# B&R Automation Studio project ACOPOStrak (part 2)

### Config_1.assembly - 5PC900_TS17_00/mappMotion/TrakOval/Config_1.assembly
```
Element gAssembly_1 (Type=assembly)
  Tracks:
    TrackSeparation = 0.030
    Track[1]:
      Segments:
        SegmentRef[1] = ::Seg_A_1
        SegmentRef[2] = ::Seg_A_2
        SegmentRef[3] = ::Seg_A_3
        SegmentRef[4] = ::Seg_A_4
        SegmentRef[5] = ::Seg_A_5
        SegmentRef[6] = ::Seg_A_6
        SegmentRef[7] = ::Seg_A_7
        SegmentRef[8] = ::Seg_A_8
        SegmentRef[9] = ::Seg_A_9
        SegmentRef[10] = ::Seg_A_10
        SegmentRef[11] = ::Seg_A_11
        SegmentRef[12] = ::Seg_A_12
        SegmentRef[13] = ::Seg_A_13
      Position = Absolute
        SegmentRef = ::Seg_A_1
        SegmentCountDirection = RightToLeft
        Translation:
          X = 0.0
          Y = 0.0
          Z = 0.0
        Orientation:
          Angle1 = 0.0
          Angle2 = 0.0
          Angle3 = 180
    Track[2]:
      Segments:
        SegmentRef[1] = ::Seg_A_14
        SegmentRef[2] = ::Seg_A_15
        SegmentRef[3] = ::Seg_A_16
        SegmentRef[4] = ::Seg_A_17
        SegmentRef[5] = ::Seg_A_18
        SegmentRef[6] = ::Seg_A_19
        SegmentRef[7] = ::Seg_A_20
        SegmentRef[8] = ::Seg_A_21
        SegmentRef[9] = ::Seg_A_22
        SegmentRef[10] = ::Seg_A_23
        SegmentRef[11] = ::Seg_A_24
        SegmentRef[12] = ::Seg_A_25
        SegmentRef[13] = ::Seg_A_26
      Position = Absolute
        SegmentRef = ::Seg_A_14
        SegmentCountDirection = RightToLeft
        Translation:
          X = 0.0
          Y = 0.0
          Z = 0.0
        Orientation:
          Angle1 = 0.0
          Angle2 = 0.0
          Angle3 = 0.0
    Track[3]:
      Segments:
        SegmentRef[1] = ::Seg_B_1
        SegmentRef[2] = :Seg_B_2
      Position = Absolute
        SegmentRef = :Seg_B_1
        SegmentCountDirection = RightToLeft
        Translation:
          X = 0.0
          Y = 0.0
          Z = 0.0
        Orientation:
          Angle1 = 0.0
          Angle2 = 0.0
          Angle3 = 0.0
    Track[4]:
      Segments:
        SegmentRef[1] = :Seg_B_3
        SegmentRef[2] = :Seg_B_4
        SegmentRef[3] = :Seg_B_5
      Position = Absolute
        SegmentRef = :Seg_B_3
        SegmentCountDirection = RightToLeft
        Translation:
          X = 0.0
          Y = 0.0
          Z = 0.0
        Orientation:
          Angle1 = 0.0
          Angle2 = 0.0
          Angle3 = 0.0
    Track[5]:
      Segments:
        SegmentRef[1] = :Seg_B_6
        SegmentRef[2] = :Seg_B_7
      Position = Absolute
        SegmentRef = :Seg_B_6
        SegmentCountDirection = RightToLeft
        Translation:
          X = 0.0
          Y = 0.0
          Z = 0.0
        Orientation:
          Angle1 = 0.0
          Angle2 = 0.0
          Angle3 = 0.0
  CommonSegmentSettings:
    SegmentSimulationOnPLC = Off
    StopReaction = InductionHalt
    SpeedFilter = NotUsed
    ControllerParameters:
      DefaultParameter:
        Controller:
          Position:
            ProportionalGain = 200
          Speed:
            ProportionalGain = 80
            IntegrationTime = 0.0
          FeedForward:
            TotalMass = 1
            ForcePositive = 0.0
            ForceNegative = 0.0
            SpeedForceFactor = 0.0
            ForceLoad = 0.0
        MovementErrorLimits:
          PositionError = 0.001
          VelocityError = 0.05
      AdditionalParameterSets = NotUsed
  Shuttles:
    MaxShuttleCount = 25
    ShuttleStereotypes:
      ShuttleStRef[1] = ShuttleStereotype_1
    MagnetPlateConfigurations:
      ShuttleType[1] = 8F1SA.100.xxxxxx-x
    CollisionAvoidance:
      Strategy = Constant
      MaximumModelDimensions:
        Length:
          ExtentToFront = 0.025
          ExtentToBack = 0.025
        Width:
          Width = 0.040
  Visualization:
    MonitoringPv = gShuttleMon
    ProcessingTaskClass = 1
```

### Config_2.shuttlestereotype - 5PC900_TS17_00/mappMotion/TrakOval/Config_2.shuttlestereotype
```
Element ShuttleStereotype_1 (Type=shuttlestereotype)
  MeasurementUnit = 5067858
  MeasurementResolution = 0.00001
  MovementLimits = Internal
    VelocityIsReadOnly = 0
    Velocity:
      Velocity = 4
    AccelerationIsReadOnly = 0
    Acceleration:
      Acceleration = 40
    DecelerationIsReadOnly = 0
    Deceleration:
      Deceleration = 40
  JerkFilter = NotUsed
  UserData:
    Size = 12
```

### Config_3.sector - 5PC900_TS17_00/mappMotion/TrakOval/Config_3.sector
```
Element SectorTrackA (Type=sector)
  Type = Composed
    StartSegment:
      SegmentRef = ::Seg_A_1
    IntermediateSegments:
      SegmentRef[1] = ::Seg_A_2
      SegmentRef[2] = ::Seg_A_3
      SegmentRef[3] = ::Seg_A_4
      SegmentRef[4] = ::Seg_A_5
      SegmentRef[5] = ::Seg_A_6
      SegmentRef[6] = ::Seg_A_7
      SegmentRef[7] = ::Seg_A_8
      SegmentRef[8] = ::Seg_A_9
      SegmentRef[9] = ::Seg_A_10
      SegmentRef[10] = ::Seg_A_11
      SegmentRef[11] = ::Seg_A_12
      SegmentRef[12] = ::Seg_A_13
      SegmentRef[13] = ::Seg_A_14
      SegmentRef[14] = ::Seg_A_15
      SegmentRef[15] = ::Seg_A_16
      SegmentRef[16] = ::Seg_A_17
      SegmentRef[17] = ::Seg_A_18
      SegmentRef[18] = ::Seg_A_19
      SegmentRef[19] = ::Seg_A_20
      SegmentRef[20] = ::Seg_A_21
      SegmentRef[21] = ::Seg_A_22
      SegmentRef[22] = ::Seg_A_23
      SegmentRef[23] = ::Seg_A_24
      SegmentRef[24] = ::Seg_A_25
    EndSegment:
      SegmentRef = ::Seg_A_26
      PositionRelativeTo = FromEnd
Element SectorPouring_1 (Type=sector)
  Type = Subsector
    SectorRef = SectorTrackA
    Start:
      Position = 0.33
    Length = 0.1
    Direction = Positive
```

### Config_5.assembly - 5PC900_TS17_00/mappMotion/TrakOval/Config_5.assembly
```
Element gAssembly_1 (Type=assembly)
  Tracks:
    TrackSeparation = 0.030
    Track[1]:
      Segments:
        SegmentRef[1] = ::Seg_A_1
        SegmentRef[2] = ::Seg_A_2
        SegmentRef[3] = ::Seg_A_3
        SegmentRef[4] = ::Seg_A_4
        SegmentRef[5] = ::Seg_A_5
        SegmentRef[6] = ::Seg_A_6
        SegmentRef[7] = ::Seg_A_7
        SegmentRef[8] = ::Seg_A_8
        SegmentRef[9] = ::Seg_A_9
        SegmentRef[10] = ::Seg_A_10
        SegmentRef[11] = ::Seg_A_11
        SegmentRef[12] = ::Seg_A_12
        SegmentRef[13] = ::Seg_A_13
        SegmentRef[14] = ::Seg_A_14
        SegmentRef[15] = ::Seg_A_15
        SegmentRef[16] = ::Seg_A_16
        SegmentRef[17] = ::Seg_A_17
        SegmentRef[18] = ::Seg_A_18
        SegmentRef[19] = ::Seg_A_19
        SegmentRef[20] = ::Seg_A_20
        SegmentRef[21] = ::Seg_A_21
        SegmentRef[22] = ::Seg_A_22
        SegmentRef[23] = ::Seg_A_23
        SegmentRef[24] = ::Seg_A_24
        SegmentRef[25] = ::Seg_A_25
        SegmentRef[26] = ::Seg_A_26
      Position = Absolute
        SegmentRef = ::Seg_A_1
        SegmentCountDirection = RightToLeft
        Translation:
          X = 0.0
          Y = 0.0
          Z = 0.0
        Orientation:
          Angle1 = 0.0
          Angle2 = 0.0
          Angle3 = 180
    Track[2]:
      Segments:
        SegmentRef[1] = ::Seg_B_3
        SegmentRef[2] = ::Seg_B_2
        SegmentRef[3] = ::Seg_B_1
      Position = RelativeToOne
        TrackSegmentPosition:
          SegmentRef = ::Seg_B_1
          Position = 0
          PositionRelativeTo = FromEnd
        Base:
          SegmentRef = ::Seg_A_1
          Position = 0.1
    Track[3]:
      Segments:
        SegmentRef[1] = ::Seg_B_4
        SegmentRef[2] = ::Seg_B_5
        SegmentRef[3] = ::Seg_B_6
        SegmentRef[4] = ::Seg_B_7
        SegmentRef[5] = ::Seg_B_8
      Position = RelativeToOne
        TrackSegmentPosition:
          SegmentRef = ::Seg_B_4
        Base:
          SegmentRef = ::Seg_B_3
          Position = 0.33
    Track[4]:
      Segments:
        SegmentRef[1] = ::Seg_B_11
        SegmentRef[2] = ::Seg_B_10
        SegmentRef[3] = ::Seg_B_9
      Position = RelativeToTwo
        AlignmentToFirst:
          SegmentRefNewFirst = ::Seg_B_11
          SegmentRefBaseFirst = ::Seg_A_7
        AlignmentToSecond:
          SegmentRefNewSecond = ::Seg_B_9
          SegmentRefBaseSecond = ::Seg_B_8
  CommonSegmentSettings:
    SegmentSimulationOnPLC = Off
    StopReaction = InductionHalt
    SpeedFilter = NotUsed
    ControllerParameters:
      DefaultParameter:
        Controller:
          Position:
            ProportionalGain = 200
          Speed:
            ProportionalGain = 80
            IntegrationTime = 0.0
          FeedForward:
            TotalMass = 1
            ForcePositive = 0.0
            ForceNegative = 0.0
            SpeedForceFactor = 0.0
            ForceLoad = 0.0
        MovementErrorLimits:
          PositionError = 0.001
          VelocityError = 0.05
      AdditionalParameterSets = NotUsed
  Shuttles:
    MaxShuttleCount = 25
    ShuttleStereotypes:
      ShuttleStRef[1] = ShuttleStereotype_1
    MagnetPlateConfigurations:
      ShuttleType[1] = 8F1SA.100.xxxxxx-x
    CollisionAvoidance:
      Strategy = Constant
      MaximumModelDimensions:
        Length:
          ExtentToFront = 0.025
          ExtentToBack = 0.025
        Width:
          Width = 0.040
  Visualization:
    MonitoringPv = gShuttleMon
    ProcessingTaskClass = 1
```

### Config_7.sector - 5PC900_TS17_00/mappMotion/TrakOval/Config_7.sector
```
Element SectorTrackA (Type=sector)
  Type = Composed
    StartSegment:
      SegmentRef = ::Seg_A_1
    IntermediateSegments:
      SegmentRef[1] = ::Seg_A_2
      SegmentRef[2] = ::Seg_A_3
      SegmentRef[3] = ::Seg_A_4
      SegmentRef[4] = ::Seg_A_5
      SegmentRef[5] = ::Seg_A_6
      SegmentRef[6] = ::Seg_A_7
      SegmentRef[7] = ::Seg_A_8
      SegmentRef[8] = ::Seg_A_9
      SegmentRef[9] = ::Seg_A_10
      SegmentRef[10] = ::Seg_A_11
      SegmentRef[11] = ::Seg_A_12
      SegmentRef[12] = ::Seg_A_13
      SegmentRef[13] = ::Seg_A_14
      SegmentRef[14] = ::Seg_A_15
      SegmentRef[15] = ::Seg_A_16
      SegmentRef[16] = ::Seg_A_17
      SegmentRef[17] = ::Seg_A_18
      SegmentRef[18] = ::Seg_A_19
      SegmentRef[19] = ::Seg_A_20
      SegmentRef[20] = ::Seg_A_21
      SegmentRef[21] = ::Seg_A_22
      SegmentRef[22] = ::Seg_A_23
      SegmentRef[23] = ::Seg_A_24
      SegmentRef[24] = ::Seg_A_25
    EndSegment:
      SegmentRef = ::Seg_A_26
      PositionRelativeTo = FromEnd
```

### Alarm.mpalarmxcore - 5PC900_TS17_00/mappServices/Alarm.mpalarmxcore
```
Element gAlarmXCore (Type=mpalarmxcore)
  mapp.AlarmX.Core.Configuration:
    [0]:
      Name = InterruptAlarm
      Message = Procces was interrupted
    [1]:
      Name = SectorTopAlarm
      Message = Top Pouring Sector inefficient
      Code = 1
      Behavior = DiscreteValueMonitoring
        Monitoring:
          MonitoredPV = ::TrakMoveme:VisPouring_Top_Broken
          TriggerValues:
            [0] = FALSE
    [2]:
      Name = SectorDownAlarm
      Message = Down Pouring Sector inefficient
      Code = 2
      Behavior = DiscreteValueMonitoring
        Monitoring:
          MonitoredPV = ::TrakMoveme:VisPouring_Down_Broken
          TriggerValues:
            [0] = FALSE
    [3]:
      Name = SuddenlyStopAlarm
      Message = Procces was suddenly stopped
    [4]:
      Name = SectorCappingAlarm
      Message = Capping Sector inefficient
      Code = 3
      Behavior = DiscreteValueMonitoring
        Monitoring:
          MonitoredPV = ::TrakMoveme:VisCapping_Broken
          TriggerValues:
            [0] = FALSE
    [5]:
      Name = SectorInputAlarm
      Message = Input Sector inefficient
      Code = 4
      Behavior = DiscreteValueMonitoring
        Monitoring:
          MonitoredPV = ::gVisInput_Broken
          TriggerValues:
            [0] = FALSE
    [6]:
      Name = SectorIOutputAlarm
      Message = Output Sector inefficient
      Code = 5
      Behavior = DiscreteValueMonitoring
        Monitoring:
          MonitoredPV = ::gVisOutput_Broken
          TriggerValues:
            [0] = FALSE
    [7]:
      Name = ManualWorkAlarm
      Message = Trak is in manual work
      Code = 6
      Severity = 10
      Behavior = DiscreteValueMonitoring
        Monitoring:
          MonitoredPV = ::TrakMoveme:VisManual
          TriggerValues:
            [0] = TRUE
    [8]:
      Name = HighAccelerationAlarm
      Message = High acceleration has been set
      Code = 7
      Severity = 10
      Behavior = LevelMonitoring
        Monitoring:
          MonitoredPV = ::TrakMoveme:VisAcceleration
          HighLimitEnable = Static
            Limit = 37
            LimitText = High acceleration has been set
    [9]:
      Name = HighDecelerationAlarm
      Message = High deceleration has been set
      Code = 9
      Severity = 10
      Behavior = LevelMonitoring
        Monitoring:
          MonitoredPV = ::TrakMoveme:VisDeceleration
          HighLimitEnable = Static
            Limit = 37
            LimitText = High deceleration has been set
    [10]:
      Name = HighVelocityAlarm
      Message = High velocity has been set
      Code = 10
      Severity = 10
      Behavior = LevelMonitoring
        Monitoring:
          MonitoredPV = ::TrakMoveme:VisVelocity
          HighLimitEnable = Static
            Limit = 3.5
            LimitText = High velocity has been set
```

## Logical view

Binary libraries used (declarations not repeated): operator, runtime, astime, AsIecCon, CoTrace, AsZip, FileIO, McBase, McAxis, McAcpTrak 5.10.1, AsBrStr, MpRobotics 5.10.1, MpBase, McAxGroup, McPathGen, McProgInt, McAcpAx, MpRecipe 5.10.1, standard, sys_lib, MpAlarmX, MpFile 5.10.1, MpServer

### Global.typ - Global data types
```iecst
(*shuttle-UserData structure*)

TYPE
	ShuttleUserData_typ : 	STRUCT
		Color : ShuttleColor_enum; (*example: product colour*)
		Weight : REAL; (*example: product weight*)
		Partnumber : UDINT; (*example: product part number*)
	END_STRUCT;
	ShuttleColor_enum :
		(
		ORANGE,
		GREEN,
		RED,
		BLUE,
		WHITE
		);
END_TYPE

(*Assembly Interface Type*)

TYPE
	TrakAsmCommand_type : 	STRUCT
		Power : BOOL;
		ShuttleStart : BOOL;
		ShuttleStop : BOOL;
	END_STRUCT;
	TrakAsmParameter_type : 	STRUCT
		Velocity : REAL;
		Acceleration : REAL;
		Deceleration : REAL;
	END_STRUCT;
	TrakAsmStatus_type : 	STRUCT
		Disabled : BOOL;
		Ready : BOOL;
		Homing : BOOL;
		Stopping : BOOL;
		ErrorStop : BOOL;
	END_STRUCT;
	TrakAsm_type : 	STRUCT
		Command : TrakAsmCommand_type;
		Parameter : TrakAsmParameter_type;
		Status : TrakAsmStatus_type;
	END_STRUCT;
	Order_type : 	STRUCT
		numberOfPackages : USINT := 5;
		bottlesPerPackage : USINT := 5;
		bottleSize : BottleSize_enum := BOTTLE_SIZE_LARGE;
		drinkColor : DrinkColor_enum := DRINK_COLOR_RED;
	END_STRUCT;
	DrinkColor_enum :
		(
		DRINK_COLOR_RED,
		DRINK_COLOR_GREEN,
		DRINK_COLOR_BLUE
		);
	BottleSize_enum :
		(
		BOTTLE_SIZE_LARGE,
		BOTTLE_SIZE_SMALL
		);
END_TYPE
```

### Global.var - Global variables
```iecst
VAR
	VisManual : BOOL;
	gbottlesDone : BOOL;
	gPartyOn : BOOL;
	gVisTurn_Broken : BOOL;
	ShuttleNumber : USINT;
END_VAR
(*Assembly interface*)
VAR
	gBottleInPlace_Turn : BOOL;
	gShuttleInPlace_Turn : BOOL;
	gTrakAsm : TrakAsm_type;
END_VAR
(*shuttle-UserData structure*)
VAR
	gShuttleUserData : ShuttleUserData_typ;
END_VAR
(*shuttle monitor structure for Vis*)
VAR
	gShuttleMon : McAcpTrakAssemblyMonData;
END_VAR
(*Bottle input and output*)
VAR
	gBottleInPlace_Input : BOOL := FALSE;
	gBottleInPlace_Output : BOOL := FALSE;
	gShuttleInPlace_Output : BOOL := FALSE;
	gShuttleInPlace_Input : BOOL := FALSE;
END_VAR
(*Trak Variables*)
VAR CONSTANT
	MAX_NUM_SHUTTLES : USINT := 25;
END_VAR
VAR
	ActiveShuttle : INT := NUM_SIM_SHUTTLES;
END_VAR
VAR CONSTANT
	NUM_SIM_SHUTTLES : USINT := 10;
END_VAR
VAR
	gShuttleColor : ARRAY[0..NUM_SIM_SHUTTLES] OF INT;
	gShuttleColored : ARRAY[0..NUM_SIM_SHUTTLES] OF BOOL;
	gColorBlue : INT;
	gColorGreen : INT;
	gColorRed : INT;
	gOrderedBottles : USINT;
	gBottlesOut : USINT;
	gColorSum : INT;
	gdiStart : BOOL;
	gOrder : Order_type;
	gVisPower : BOOL;
	gCurrentRecipeName : STRING[255];
	gProcessFinished : BOOL;
	gdiStop : BOOL;
	gVisOutput_Broken : BOOL := TRUE;
	gVisInput_Broken : BOOL := TRUE;
	gBgColor : ARRAY[0..2] OF REAL;
	gDeltaVelocity : USINT := 100;
	gdiInstantStop : BOOL;
	VisDeltaVelocity : REAL := 0.0;
	VisDeltaInJogXAdd : BOOL;
	VisDeltaInJogXSub : BOOL;
	VisDeltaInJogYAdd : BOOL;
	VisDeltaInJogYSub : BOOL;
	VisDeltaInJogZAdd : BOOL;
	VisDeltaInJogZSub : BOOL;
	BottleOutStage : USINT;
	BottleInStage : USINT;
	Bottle : INT;
	VisDeltaNumber : USINT;
END_VAR
```

### Package Logical/Libraries - Global libraries

- Visualisation Logical/mappView (not shown)

### Program Logical/svgTransform (IEC)

#### Types.typ
```iecst
TYPE
	stationName :
		(
		Input,
		Output,
		NozzleUp,
		TwistOn,
		NozzleDown
		);
END_TYPE
```

#### Variables.var
```iecst
VAR
	tranformation : STRING[255];
	loopTmp : USINT;
	svgBlocksToColor : ARRAY[0..5] OF USINT;
END_VAR
```

#### Main.st
```iecst
PROGRAM _INIT
	(* Insert code here *)
	loopTmp := 1;
	ShuttleNumber :=1;
END_PROGRAM

PROGRAM _CYCLIC
	// 0 -> włączony
	// 1 -> error
	// 2 -> wyłączony

	CASE loopTmp OF
		1:
			//WEJŚCIE
			IF svgBlocksToColor[0] = 0 THEN
				tranformation := '[{"select":"#wejscie","duration":500,"fill":1}]';
			ELSIF svgBlocksToColor[0] = 1 THEN
				tranformation := '[{"select":"#wejscie","duration":500,"fill":2}]';
			ELSIF svgBlocksToColor[0] = 2 THEN
				tranformation := '[{"select":"#wejscie","duration":500,"fill":3}]';
			END_IF;
		2:
			//WYJŚCIE
			IF svgBlocksToColor[1] = 0 THEN
				tranformation := '[{"select":"#wyjscie","duration":500,"fill":1}]';
			ELSIF svgBlocksToColor[1] = 1 THEN
				tranformation := '[{"select":"#wyjscie","duration":500,"fill":2}]';
			ELSIF svgBlocksToColor[1] = 2 THEN
				tranformation := '[{"select":"#wyjscie","duration":500,"fill":3}]';
			END_IF;
		3:
			//ZAKRĘCANIE
			IF svgBlocksToColor[2] = 0 THEN
				tranformation := '[{"select":"#zakrecanie","duration":500,"fill":1}]';
			ELSIF svgBlocksToColor[2] = 1 THEN
				tranformation := '[{"select":"#zakrecanie","duration":500,"fill":2}]';
			ELSIF svgBlocksToColor[2] = 2 THEN
				tranformation := '[{"select":"#zakrecanie","duration":500,"fill":3}]';
			END_IF;
		4:
			//NALEWANIE A(dół)
			IF svgBlocksToColor[3] = 0 THEN
				tranformation := '[{"select":"#nalewanieA","duration":500,"fill":1}]';
			ELSIF svgBlocksToColor[3] = 1 THEN
				tranformation := '[{"select":"#nalewanieA","duration":500,"fill":2}]';
			ELSIF svgBlocksToColor[3] = 2 THEN
				tranformation := '[{"select":"#nalewanieA","duration":500,"fill":3}]';
			END_IF;
		5:
			//NALEWANIE B(góra)
			IF svgBlocksToColor[4] = 0 THEN
				tranformation := '[{"select":"#nalewanieB","duration":500,"fill":1}]';
			ELSIF svgBlocksToColor[4] = 1 THEN
				tranformation := '[{"select":"#nalewanieB","duration":500,"fill":2}]';
			ELSIF svgBlocksToColor[4] = 2 THEN
				tranformation := '[{"select":"#nalewanieB","duration":500,"fill":3}]';
			END_IF;
	END_CASE;

	IF loopTmp = 5 THEN
		loopTmp := 1;
	ELSE
		loopTmp := loopTmp + 1;
	END_IF;
END_PROGRAM

PROGRAM _EXIT
	(* Insert code here *)
END_PROGRAM
```

### Program Logical/Robots/DeltaIn (IEC)

#### Main.st - Init, cyclic, exit code
```iecst
PROGRAM _INIT

	MpDelta3Axis_0.MpLink := ADR(g3AxDeltaA);
	MpDelta3Axis_0.Enable := TRUE;
	MpDelta3Axis_0.Parameters := ADR(DeltaParameters);

	MpDelta3Axis_0.Override := 100.0;
	DeltaParameters.Velocity := 5.0;
	DeltaParameters.Acceleration := 50.0;
	Step := INIT;
	VisManual:=FALSE;
	BottleInStage:=0;
END_PROGRAM

PROGRAM _CYCLIC

	MpDelta3Axis_0.Override:=gDeltaVelocity;

	IF gdiInstantStop THEN
		Step:=STOP;
	END_IF;

	IF EDGEPOS(MpDelta3Axis_0.Error) THEN
		Step := ERROR;
	END_IF;
	IF VisManual THEN
		Step:=MANUAL;
		END_IF
	CASE Step OF
		INIT:
			MpDelta3Axis_0.Power := FALSE;
			MpDelta3Axis_0.Home := FALSE;
			MpDelta3Axis_0.MoveProgram := FALSE;
			IF gVisPower THEN
				Step := POWER;
			END_IF;
		POWER:
			MpDelta3Axis_0.Power := TRUE;
			VisDeltaInState:=1;
			IF MpDelta3Axis_0.PowerOn THEN
				Step:= HOME;
			END_IF;
		HOME:
			MpDelta3Axis_0.Home := TRUE;
			IF MpDelta3Axis_0.IsHomed THEN
				Step := WAIT_SHUTTLE;

			END_IF;
		WAIT_SHUTTLE:
			BottleInStage:=0;
			IF MpDelta3Axis_0.Home=FALSE  THEN
				MpDelta3Axis_0.Home:=TRUE;
			END_IF;
			VisDeltaInState:=2;
			MpDelta3Axis_0.MoveProgram := 0;
			IF gShuttleInPlace_Input AND NOT gdiStop  THEN
				Step := MOVE_PROGRAM;
				DeltaParameters.ProgramName := 'RoboticIn.st';    //File stored on FileDevice
			END_IF;

		MOVE_PROGRAM:
			IF MpDelta3Axis_0.Z=-700 AND MpDelta3Axis_0.Y=-200 THEN
	  			BottleInStage:=1;
			END_IF;
			IF MpDelta3Axis_0.Z=-700 AND MpDelta3Axis_0.Y=200 THEN
				BottleInStage:=2;
			END_IF;
			VisDeltaInState:=3;
			IF gVisInput_Broken THEN
				IF gColorSum >0 THEN
					MpDelta3Axis_0.MoveProgram :=TRUE;
					IF MpDelta3Axis_0.MoveDone THEN
						gColorSum := gColorSum - 1;
						Step:= WAIT_SHUTTLE;
						gBottleInPlace_Input:=TRUE;

					END_IF;
					IF diInterrupt THEN
						Step := INTERRUPT;
						MpDelta3Axis_0.Continue := FALSE;
					END_IF;
				END_IF;
			ELSE
				Step := INTERRUPT;
				MpDelta3Axis_0.Continue := FALSE;

			END_IF;
			IF gTrakAsm.Command.Power=FALSE THEN
				Step:=STOP;
			END_IF;

		INTERRUPT:
			VisDeltaInState:=4;
			MpDelta3Axis_0.Interrupt := TRUE;
			IF NOT (diInterrupt) OR EDGEPOS(gVisInput_Broken) THEN
				MpDelta3Axis_0.Interrupt := FALSE;
				MpDelta3Axis_0.Continue := TRUE;
				Step := MOVE_PROGRAM;
			END_IF;

		STOP:
			MpDelta3Axis_0.Stop := TRUE;
			IF (NOT gdiInstantStop) AND MpDelta3Axis_0.Stopped THEN
				MpDelta3Axis_0.Home := FALSE;
				MpDelta3Axis_0.Interrupt := FALSE;
				MpDelta3Axis_0.Continue := FALSE;
				MpDelta3Axis_0.MoveProgram := FALSE;
				MpDelta3Axis_0.Stop := FALSE;
				Step := INIT;
			END_IF;
		ERROR:
			MpDelta3Axis_0.MoveProgram := FALSE;
			MpDelta3Axis_0.ErrorReset := TRUE;

			IF NOT(MpDelta3Axis_0.Error) THEN
				Step := WAIT_SHUTTLE;
				MpDelta3Axis_0.ErrorReset := FALSE;
			END_IF;

		MANUAL:
			MpDelta3Axis_0.Override:=100;
			gDeltaVelocity:=100;
			MpDelta3Axis_0.Jog:=TRUE;
			IF VisDeltaNumber = 0 THEN
				IF VisDeltaInJogXAdd THEN
					DeltaParameters.Jog.Velocity[0]:=VisDeltaVelocity;
				END_IF;
				IF EDGENEG(VisDeltaInJogXAdd) THEN
					DeltaParameters.Jog.Velocity[0]:=0.0;
				END_IF;
				IF VisDeltaInJogXSub THEN
					DeltaParameters.Jog.Velocity[0]:=-VisDeltaVelocity;
				END_IF;
				IF EDGENEG(VisDeltaInJogXSub) THEN
					DeltaParameters.Jog.Velocity[0]:=0.0;
				END_IF;
				IF VisDeltaInJogYAdd THEN
					DeltaParameters.Jog.Velocity[1]:=VisDeltaVelocity;
				END_IF;
				IF EDGENEG(VisDeltaInJogYAdd) THEN
					DeltaParameters.Jog.Velocity[1]:=0.0;
				END_IF;
				IF VisDeltaInJogYSub THEN
					DeltaParameters.Jog.Velocity[1]:=-VisDeltaVelocity;
				END_IF;
				IF EDGENEG(VisDeltaInJogYSub) THEN
					DeltaParameters.Jog.Velocity[1]:=0.0;
				END_IF;
				IF VisDeltaInJogZAdd THEN
					DeltaParameters.Jog.Velocity[2]:=VisDeltaVelocity;
				END_IF;
				IF EDGENEG(VisDeltaInJogZAdd) THEN
					DeltaParameters.Jog.Velocity[2]:=0.0;
				END_IF;
				IF VisDeltaInJogZSub THEN
					DeltaParameters.Jog.Velocity[2]:=-VisDeltaVelocity;
				END_IF;
				IF EDGENEG(VisDeltaInJogZSub) THEN
					DeltaParameters.Jog.Velocity[2]:=0.0;
				END_IF;
			END_IF;

			IF gTrakAsm.Command.Power=FALSE THEN
				Step:=STOP;
			END_IF;

	END_CASE;
	IF Step=MANUAL AND VisManual=FALSE THEN
		MpDelta3Axis_0.Jog:=FALSE;
		IF MpDelta3Axis_0.Home=FALSE THEN
			//MpDelta3Axis_0.Home:=TRUE;
			Step:=WAIT_SHUTTLE;
		ELSE
			MpDelta3Axis_0.Home:=FALSE;
		END_IF;
	END_IF;
		MpDelta3Axis_0();
	END_PROGRAM

PROGRAM _EXIT

	MpDelta3Axis_0.Power  := FALSE;
	MpDelta3Axis_0.Home   := FALSE;
	MpDelta3Axis_0.MoveDirect := FALSE;
	MpDelta3Axis_0.MoveLinear := FALSE;
	MpDelta3Axis_0();

	MpDelta3Axis_0.Enable := FALSE;
	MpDelta3Axis_0();

				END_PROGRAM
```

#### Variables.var - Local variables
```iecst
VAR
	VisDeltaInState : USINT;
	MpDelta3Axis_0 : MpDelta3Axis;
	DeltaParameters : MpDelta3AxisParType;
	Step : StepType;
	diInterrupt : BOOL := FALSE;
	ZOffset : LREAL;
	DeltaInBottleVisibility : BOOL;
	DeltaInBottleShutVis : BOOL;
END_VAR
```

### Program Logical/Robots/DeltaOut (IEC)

#### Main.st - Init, cyclic, exit code
```iecst
PROGRAM _INIT

	MpDelta3Axis_0.MpLink := ADR(g3AxDeltaAOut);
	MpDelta3Axis_0.Enable := TRUE;
	MpDelta3Axis_0.Parameters := ADR(DeltaParameters);

	MpDelta3Axis_0.Override := 100.0;

	DeltaParameters.ProgramName:='RoboticOut.st';
	DeltaParameters.Velocity := 5.0;
	DeltaParameters.Acceleration := 50.0;
	BottleOutStage:=0;
END_PROGRAM

PROGRAM _CYCLIC
	MpDelta3Axis_0.Override:=gDeltaVelocity;
	//DeltaParameters.ProgramName := PName;
	MpDelta3Axis_0.ErrorReset := diErrorReset;

	IF EDGEPOS(MpDelta3Axis_0.Error) THEN
		Step := ERROR;
	END_IF;
	IF VisManual THEN
		Step:=MANUAL;
	END_IF

	CASE Step OF
		INIT:
			MpDelta3Axis_0.Power := FALSE;
			MpDelta3Axis_0.Home := FALSE;
			MpDelta3Axis_0.MoveProgram := FALSE;

			IF gVisPower THEN
				Step := POWER;
			END_IF;
		POWER:
			MpDelta3Axis_0.Power := TRUE;
			VisDeltaOutState:=1;
			IF MpDelta3Axis_0.PowerOn THEN
				Step := HOME;
			END_IF;
		HOME:
			MpDelta3Axis_0.Home := TRUE;

			IF MpDelta3Axis_0.IsHomed THEN
				Step := WAIT_SHUTTLE;
			END_IF;
		WAIT_SHUTTLE:
			BottleOutStage:=0;
			IF MpDelta3Axis_0.Home=FALSE  THEN
				MpDelta3Axis_0.Home:=TRUE;
			END_IF;
			VisDeltaOutState:=2;
			IF ProgressBar > 99 AND diStart THEN
				gBottlesDone := 0;
				ProgressBar := 0;
			END_IF;

			IF gShuttleInPlace_Output THEN
				Step := MOVE_PROGRAM;
				gBottlesDone := gBottlesDone+1;
				ProgressBar := 100*gBottlesDone/gOrder.bottlesPerPackage/gOrder.numberOfPackages;
			END_IF;
			IF gTrakAsm.Command.Power=FALSE THEN
				Step:=STOP;
			END_IF;
		MOVE_PROGRAM:
			IF MpDelta3Axis_0.Z=-700 AND MpDelta3Axis_0.Y=200 THEN
				BottleOutStage:=1;
			END_IF;
			IF NOT(MpDelta3Axis_0.Z=-700 AND MpDelta3Axis_0.Y=200) AND MpDelta3Axis_0.PathVelocity=0 AND BottleOutStage=1 THEN
				BottleOutStage:=2;
			END_IF;
			diStart := FALSE;
			VisDeltaOutState:=3;
			IF gVisOutput_Broken THEN
				IF gOrder.bottlesPerPackage = 4 THEN
					CASE BottlesPerPack OF

						1:	Bottle:=1;

						2:	Bottle:=2;

						3:	Bottle:=5;

						4:	Bottle:=4;

					END_CASE;
				ELSE
					CASE BottlesPerPack OF

						1:	Bottle:=1;

						2:	Bottle:=2;

						3:	Bottle:=3;

						4:	Bottle:=4;

						5:	Bottle:=5;

						6:	Bottle:=6;

					END_CASE;
				END_IF;
				MpDelta3Axis_0.MoveProgram := TRUE;
				IF MpDelta3Axis_0.MoveDone THEN
					BottlesPerPack:=BottlesPerPack+1;
					MpDelta3Axis_0.MoveProgram := FALSE;
					Step := WAIT_SHUTTLE;
					gBottleInPlace_Output:=TRUE;
					BottleOutStage:=0;
					IF BottlesPerPack>gOrder.bottlesPerPackage THEN
						BottlesPerPack:=1;
					END_IF;

				END_IF;
			ELSE
				Step := INTERRUPT;
				MpDelta3Axis_0.Continue := FALSE;
			END_IF;
			IF gTrakAsm.Command.Power=FALSE THEN
				Step:=STOP;
			END_IF;
		INTERRUPT:
			MpDelta3Axis_0.Interrupt := TRUE;
			VisDeltaOutState:=4;
			IF EDGEPOS (gVisOutput_Broken) THEN
				MpDelta3Axis_0.Interrupt := FALSE;
				MpDelta3Axis_0.Continue := TRUE;
				Step := MOVE_PROGRAM;
			END_IF;
		STOP:
			MpDelta3Axis_0.Stop := TRUE;
			IF (NOT gdiInstantStop) AND MpDelta3Axis_0.Stopped THEN

				MpDelta3Axis_0.Home := FALSE;
				MpDelta3Axis_0.Interrupt := FALSE;
				MpDelta3Axis_0.Continue := FALSE;
				MpDelta3Axis_0.MoveProgram := FALSE;
				MpDelta3Axis_0.Stop := FALSE;

				Step := INIT;
			END_IF;
		ERROR:

			MpDelta3Axis_0.MoveProgram := FALSE;
			MpDelta3Axis_0.ErrorReset := TRUE;

			IF NOT(MpDelta3Axis_0.Error) THEN
				Step := WAIT_SHUTTLE;
				MpDelta3Axis_0.ErrorReset := FALSE;
			END_IF;

		MANUAL:
			MpDelta3Axis_0.Override:=100;
			gDeltaVelocity:=100;
			MpDelta3Axis_0.Jog:=TRUE;
			IF VisDeltaNumber = 1 THEN
				IF VisDeltaInJogXAdd THEN
					DeltaParameters.Jog.Velocity[0]:=VisDeltaVelocity;
				END_IF;
				IF EDGENEG(VisDeltaInJogXAdd) THEN
					DeltaParameters.Jog.Velocity[0]:=0.0;
				END_IF;
				IF VisDeltaInJogXSub THEN
					DeltaParameters.Jog.Velocity[0]:=-VisDeltaVelocity;
				END_IF;
				IF EDGENEG(VisDeltaInJogXSub) THEN
					DeltaParameters.Jog.Velocity[0]:=0.0;
				END_IF;
				IF VisDeltaInJogYAdd THEN
					DeltaParameters.Jog.Velocity[1]:=VisDeltaVelocity;
				END_IF;
				IF EDGENEG(VisDeltaInJogYAdd) THEN
					DeltaParameters.Jog.Velocity[1]:=0.0;
				END_IF;
				IF VisDeltaInJogYSub THEN
					DeltaParameters.Jog.Velocity[1]:=-VisDeltaVelocity;
				END_IF;
				IF EDGENEG(VisDeltaInJogYSub) THEN
					DeltaParameters.Jog.Velocity[1]:=0.0;
				END_IF;
				IF VisDeltaInJogZAdd THEN
					DeltaParameters.Jog.Velocity[2]:=VisDeltaVelocity;
				END_IF;
				IF EDGENEG(VisDeltaInJogZAdd) THEN
					DeltaParameters.Jog.Velocity[2]:=0.0;
				END_IF;
				IF VisDeltaInJogZSub THEN
					DeltaParameters.Jog.Velocity[2]:=-VisDeltaVelocity;
				END_IF;
				IF EDGENEG(VisDeltaInJogZSub) THEN
					DeltaParameters.Jog.Velocity[2]:=0.0;
				END_IF;
			END_IF;
			IF gTrakAsm.Command.Power=FALSE THEN
				Step:=STOP;
			END_IF;

	END_CASE;
	IF Step=MANUAL AND VisManual=FALSE THEN
		MpDelta3Axis_0.Jog:=FALSE;
		IF MpDelta3Axis_0.Home=FALSE THEN
			//MpDelta3Axis_0.Home:=TRUE;
			Step:=WAIT_SHUTTLE;
		ELSE
			MpDelta3Axis_0.Home:=FALSE;
		END_IF;
	END_IF;

	MpDelta3Axis_0();

END_PROGRAM

PROGRAM _EXIT

	MpDelta3Axis_0.Power  := FALSE;
	MpDelta3Axis_0.Home   := FALSE;
	MpDelta3Axis_0.MoveDirect := FALSE;
	MpDelta3Axis_0.MoveLinear := FALSE;
	MpDelta3Axis_0();

	MpDelta3Axis_0.Enable := FALSE;
	MpDelta3Axis_0();

END_PROGRAM
```

#### Variables.var - Local variables
```iecst
(*FB's*)
VAR
	DeltaParameters : MpDelta3AxisParType;
	MpDelta3Axis_0 : MpDelta3Axis;
END_VAR
(*IO's*)
VAR
	diErrorReset : BOOL;
END_VAR
(*Other*)
VAR
	Step : StepType;
	BottlesPerPack : USINT := 1;
	ProgressBar : INT;
	gBottlesDone : INT;
	diStart : BOOL;
	VisDeltaOutState : USINT;
	DeltaOutBottleVisibility : BOOL;
	StashBottleVis : ARRAY[0..5] OF BOOL;
	i : INT;
	DeltaOutBottleShutVis : BOOL;
	ZOffset : LREAL;
	BottleInvisible : BOOL;
END_VAR
```

### Types.typ
```iecst
TYPE
	StepType :
		(
		INIT,
		POWER,
		HOME,
		WAIT_SHUTTLE,
		MOVE_PROGRAM,
		INTERRUPT,
		MANUAL,
		STOP,
		ERROR
		);
END_TYPE
```

### Program Logical/Robots/SI (IEC)

#### Main.st - Init, cyclic, exit code
```iecst
PROGRAM _INIT

	MpDelta3Axis_0.MpLink := ADR(g3AxDeltaA_SI);
	MpDelta3Axis_0.Enable := TRUE;
	MpDelta3Axis_0.Parameters := ADR(MpDelta3AxisPar_0);

	MpDelta3Axis_0.Override := 100.0;

	MpDelta3AxisPar_0.Velocity := 5.0;
	MpDelta3AxisPar_0.Acceleration := 50.0;

	MpDelta3AxisPar_0.ProgramName := 'SI.st';

END_PROGRAM

PROGRAM _CYCLIC

	//DeltaParameters.ProgramName := PName;
	MpDelta3Axis_0();

	IF EDGEPOS(MpDelta3Axis_0.Error) THEN
		Step := ERROR;
	END_IF;

	CASE Step OF
		INIT:
			MpDelta3Axis_0.Power := FALSE;
			MpDelta3Axis_0.Home := FALSE;
			MpDelta3Axis_0.MoveProgram := FALSE;

			IF gVisPower THEN
				Step := POWER;
			END_IF;
		POWER:
			MpDelta3Axis_0.Power := TRUE;

			IF MpDelta3Axis_0.PowerOn THEN
				Step := HOME;
			END_IF;
		HOME:
			MpDelta3Axis_0.Home := TRUE;

			IF MpDelta3Axis_0.IsHomed THEN
				Step := WAIT_SHUTTLE;
			END_IF;
		WAIT_SHUTTLE:

			IF gPartyOn THEN
				Step := MOVE_PROGRAM;
			ELSE
				x := 0;
				y := 0;
				z := 0;
			END_IF;
			//RecipeBottlesPerPack := gOrder.bottlesPerPackage;
		MOVE_PROGRAM:
			MpDelta3Axis_0.MoveProgram := TRUE;

			IF MpDelta3Axis_0.MoveDone THEN
				MpDelta3Axis_0.MoveProgram := FALSE;
				Step := WAIT_SHUTTLE;
			END_IF;

			IF x=360 THEN

				IF y=360 THEN
					z := z+4;
					IF z=360 THEN
						x := 0;
						y := 0;
						z := 0;
					END_IF;
				ELSE
					y := y+4;
				END_IF;
			ELSE
				x := x+4;
			END_IF;

	END_CASE;

	MpDelta3Axis_0();

END_PROGRAM

PROGRAM _EXIT

	MpDelta3Axis_0.Power  := FALSE;
	MpDelta3Axis_0.Home   := FALSE;
	MpDelta3Axis_0.MoveDirect := FALSE;
	MpDelta3Axis_0.MoveLinear := FALSE;
	MpDelta3Axis_0();

	MpDelta3Axis_0.Enable := FALSE;
	MpDelta3Axis_0();

END_PROGRAM
```

#### Variables.var - Local variables
```iecst
VAR
	MpDelta3AxisPar_0 : MpDelta3AxisParType;
	MpDelta3Axis_0 : MpDelta3Axis;
	Step : StepType;
	x : INT;
	y : INT;
	z : INT;
END_VAR
```

### Program Logical/Robots/DeltaTurn

#### Variables.var
```iecst
VAR
	DeltaParameters : MpDelta4AxisParType;
	MpDelta4Axis_0 : MpDelta4Axis;
	Step : StepType;
	diErrorReset : BOOL;
	turned : UINT;
END_VAR
```

#### Main.st
```iecst
PROGRAM _INIT
	(* Insert code here *)
	MpDelta4Axis_0.MpLink := ADR(g4AxDeltaA);
	MpDelta4Axis_0.Enable := TRUE;
	MpDelta4Axis_0.Parameters := ADR(DeltaParameters);

	MpDelta4Axis_0.Override := 100.0;
	DeltaParameters.ProgramName := 'RoboticDown.st';    //File stored on FileDevice

	DeltaParameters.Velocity := 5.0;
	DeltaParameters.Acceleration := 50.0;

	DeltaParameters.Jog.Velocity[3] := 100;

	Step :=INIT;

END_PROGRAM

PROGRAM _CYCLIC
	(* Insert code here *)
	MpDelta4Axis_0();

	IF gdiInstantStop THEN
		Step:=STOP;
	END_IF;

	MpDelta4Axis_0.ErrorReset := diErrorReset;
	IF EDGEPOS(MpDelta4Axis_0.Error) THEN
		Step := ERROR;
	END_IF;

	CASE Step OF
		INIT:
			MpDelta4Axis_0.Power := FALSE;
			MpDelta4Axis_0.Home := FALSE;
			MpDelta4Axis_0.MoveProgram := FALSE;
			IF gVisPower THEN
				Step := POWER;
			END_IF;
		POWER:
			MpDelta4Axis_0.Power := TRUE;
			IF MpDelta4Axis_0.PowerOn THEN
				Step:= HOME;
			END_IF;
		HOME:
			MpDelta4Axis_0.Home := TRUE;
			IF MpDelta4Axis_0.IsHomed THEN
				Step := WAIT_SHUTTLE;
			END_IF;
		WAIT_SHUTTLE:
			MpDelta4Axis_0.MoveProgram := FALSE;
			IF EDGEPOS(gShuttleInPlace_Turn) THEN
				Step := MOVE_PROGRAM;
			END_IF;
			turned := 0;

		MOVE_PROGRAM:
			IF NOT(gVisTurn_Broken) THEN
					MpDelta4Axis_0.MoveProgram :=TRUE;

					//Turning the robot around
					IF turned<240 THEN
						turned := turned+8;
					END_IF;

					IF MpDelta4Axis_0.MoveDone THEN
						Step:= WAIT_SHUTTLE;
						gBottleInPlace_Turn:=TRUE;
						gShuttleInPlace_Turn := FALSE;
					END_IF;
				ELSE
					Step := INTERRUPT;
					MpDelta4Axis_0.Continue := FALSE;
			END_IF;
		INTERRUPT:
			MpDelta4Axis_0.Interrupt := TRUE;
			IF EDGEPOS(gVisTurn_Broken) THEN
				MpDelta4Axis_0.Interrupt := FALSE;
				MpDelta4Axis_0.Continue := TRUE;
				Step := MOVE_PROGRAM;
			END_IF;

		STOP:
			MpDelta4Axis_0.Stop := TRUE;
			IF (NOT gdiInstantStop) AND MpDelta4Axis_0.Stopped THEN

				MpDelta4Axis_0.Home := FALSE;
				MpDelta4Axis_0.Interrupt := FALSE;
				MpDelta4Axis_0.Continue := FALSE;
				MpDelta4Axis_0.MoveProgram := FALSE;
				MpDelta4Axis_0.Stop := FALSE;

				Step := INIT;
			END_IF;
		ERROR:

			MpDelta4Axis_0.MoveProgram := FALSE;
			MpDelta4Axis_0.ErrorReset := TRUE;

			IF NOT(MpDelta4Axis_0.Error) THEN
				Step := WAIT_SHUTTLE;
				MpDelta4Axis_0.ErrorReset := FALSE;
			END_IF;

	END_CASE;
END_PROGRAM

PROGRAM _EXIT
	(* Insert code here *)
	MpDelta4Axis_0.Power  := FALSE;
	MpDelta4Axis_0.Home   := FALSE;
	MpDelta4Axis_0.MoveDirect := FALSE;
	MpDelta4Axis_0.MoveLinear := FALSE;
	MpDelta4Axis_0();

	MpDelta4Axis_0.Enable := FALSE;
	MpDelta4Axis_0();
END_PROGRAM
```

### Program Logical/Trak/TrakMovement (IEC)

#### Types.typ
```iecst
TYPE
	StepEnum :
		(
		POWER_OFF,
		POWER_ON,
		ADD_SHUTTLE,
		GET_SHUTTLE,
		READY,
		PROCESS,
		STOPPING,
		RESET,
		MANUAL,
		DELTA_TURN,
		DELTA_MOVE
		);
	StepSector :
		(
		Bottle_Input,
		WaitPour,
		Pouring_Down,
		Pouring_Top,
		WaitCap,
		Capping,
		Bottle_Output
		);
END_TYPE
```

#### Variables.var
```iecst
VAR
	SimShuttlePosition : ARRAY[1..MAX_NUM_SHUTTLES] OF LREAL;
END_VAR
(*sequence control*)
VAR
	Step : StepEnum;
	Step_Sector : StepSector;
	ShuttleAxis : ARRAY[1..MAX_NUM_SHUTTLES] OF McAxisType;
	CntShuttle : UINT;
	i : INT;
	DeltaInit : BOOL := FALSE;
	DeltaFor : USINT;
	Delta_Shuttle : USINT := 0;
END_VAR
(*FUB*)
VAR
	MC_BR_AsmPowerOn_AcpTrak_0 : MC_BR_AsmPowerOn_AcpTrak;
	MC_BR_AsmPowerOff_AcpTrak_0 : MC_BR_AsmPowerOff_AcpTrak;
	MC_BR_SecAddShuttle_AcpTrak_0 : MC_BR_SecAddShuttle_AcpTrak;
	MC_BR_AsmGetShuttle_AcpTrak_0 : MC_BR_AsmGetShuttle_AcpTrak;
	MC_BR_RoutedMoveVel_AcpTrak_0 : MC_BR_RoutedMoveVel_AcpTrak;
	MC_BR_RoutedMoveAbs_AcpTrak_0 : MC_BR_RoutedMoveAbs_AcpTrak;
	MC_BR_AsmReadStatus_AcpTrak_0 : MC_BR_AsmReadStatus_AcpTrak;
	MC_BR_AsmReset_AcpTrak_0 : MC_BR_AsmReset_AcpTrak;
	MC_BR_ShReadInfo_AcpTrak_0 : MC_BR_ShReadInfo_AcpTrak;
	MC_Stop_0 : MC_Stop;
	SizeofUserdata : UDINT;
	Shuttles_exist : BOOL;
END_VAR
(*Timers*)
VAR
	TON_Pouring_Down : TON;
	TON_Pouring_Top : TON;
	TON_Capping : TON := (PT:=T#4s);
	TON_Delta : TON := (PT:=T#12s);
END_VAR
(*Pouring and Capping*)
VAR
	Pouring_Down_Busy : BOOL := FALSE;
	Pouring_Down_Comming : BOOL := FALSE;
	Pouring_Down_Broken : BOOL := FALSE;
	Pouring_Top_Busy : BOOL := FALSE;
	Pouring_Top_Comming : BOOL := FALSE;
	Pouring_Top_Broken : BOOL := FALSE;
	Capping_Busy : BOOL := FALSE;
	Stop_With_Execution : BOOL := FALSE;
	Capping_Comming : BOOL := FALSE;
	Capping_Broken : BOOL := FALSE;
	ManualShuttleReset : INT;
END_VAR
(*Visualization*)
VAR
	VisShuttleStart : BOOL := FALSE;
	VisShuttleStop : BOOL := FALSE;
	VisCapping_Broken : BOOL := TRUE;
	VisPouring_Top_Broken : BOOL := TRUE;
	VisPouring_Down_Broken : BOOL := TRUE;
	VisPouring_Time_Large : REAL := 4.0;
	VisPouring_Time_Small : REAL := 2.0;
	VisVelocity : REAL := 2.0;
	VisAcceleration : REAL := 10;
	VisDeceleration : REAL := 5;
	VisShuttle : USINT := 1;
	VisManualVelocity : REAL := 1.0;
	VisManualSectorTop : BOOL := FALSE;
	VisMove_Pos : BOOL := FALSE;
	VisMove_Neg : BOOL;
	NullOrder : BOOL := FALSE;
	VisCappingStates : USINT := 0;
	VisTrakStates : USINT;
	VisPouringStates : ARRAY[0..1] OF USINT := [2(0)];
	SvgTranform : ARRAY[0..5] OF USINT;
END_VAR
(*Visualization Bottle controll*)
VAR
	BottleMaterial : ARRAY[0..9] OF USINT;
	BottleVisibility : ARRAY[0..9] OF BOOL := [10(0)];
	Capping_Position : REAL := 450;
	Capping_Rotate : REAL := 0;
	Pouring_Top_Position : INT := 400;
	Pouring_Down_Position : INT := 400;
	VisCappingRotate : BOOL;
	VisCappingAdd : BOOL;
	VisCappingSub : BOOL;
	VisPouringNumber : INT;
	VisPouringAdd : BOOL;
	VisPouringSub : BOOL;
	ManualEnable : BOOL;
END_VAR
```

#### Main.st
```iecst
PROGRAM _INIT

	gProcessFinished := TRUE;
	gVisPower := FALSE;

	// Adding Shuttles for simulation
	FOR i := 1 TO NUM_SIM_SHUTTLES DO
		SimShuttlePosition[i] := 0.15 * (i - 1);
	END_FOR

	//   Setting init trak speed
	gTrakAsm.Parameter.Velocity := 2.0;
	gTrakAsm.Parameter.Acceleration := 20;
	gTrakAsm.Parameter.Deceleration := 20;

	//Write this value into the Size of Userdata in the Shuttle Stereotype configuration
	SizeofUserdata := SIZEOF(gShuttleUserData);

	//Assembly reference for init configuration
	MC_BR_AsmPowerOn_AcpTrak_0.Assembly     := ADR(gAssembly_1);
	MC_BR_AsmGetShuttle_AcpTrak_0.Assembly  := ADR(gAssembly_1);
	MC_BR_AsmPowerOff_AcpTrak_0.Assembly    := ADR(gAssembly_1);
	MC_BR_AsmReadStatus_AcpTrak_0.Assembly  := ADR(gAssembly_1);
	MC_BR_AsmReset_AcpTrak_0.Assembly       := ADR(gAssembly_1);

	//Enable reading of current status of the assembly
	MC_BR_AsmReadStatus_AcpTrak_0.Enable := TRUE;

	// Setting timer for Pouring_Down/Up and Capping
	TON_Pouring_Top.IN:=FALSE;
	TON_Pouring_Down.IN:=FALSE;
	TON_Capping.IN:=FALSE;

END_PROGRAM

PROGRAM _CYCLIC

	// Turn off Shuttle read info and execute it
	MC_BR_ShReadInfo_AcpTrak_0.Enable     :=FALSE;
	MC_BR_ShReadInfo_AcpTrak_0();

	// Turn off absolute movement of Shuttle and execute it
	MC_BR_RoutedMoveAbs_AcpTrak_0.Execute := FALSE;
	MC_BR_RoutedMoveAbs_AcpTrak_0();
	MC_BR_RoutedMoveVel_AcpTrak_0.Execute:=FALSE;
	MC_BR_RoutedMoveVel_AcpTrak_0();
	CASE Step OF

		// Assemply power off and waiting for power on command
		POWER_OFF:
			VisTrakStates:=0;
			// When power off is done, delete the shuttle reference
			IF EDGEPOS(MC_BR_AsmPowerOff_AcpTrak_0.Done) THEN
				MC_BR_AsmPowerOff_AcpTrak_0.Execute := FALSE;
				brsmemset(ADR(ShuttleAxis), 0, SIZEOF(ShuttleAxis));
				// Assembly is not powered off yet
			ELSIF NOT(gTrakAsm.Status.Disabled) THEN
				MC_BR_AsmPowerOff_AcpTrak_0.Execute := TRUE;
			ELSIF (gTrakAsm.Command.Power) THEN
				Step := POWER_ON;
			END_IF

			// Assembly power ON
		POWER_ON:
			VisTrakStates:=1;
			MC_BR_AsmPowerOn_AcpTrak_0.Execute := TRUE;

			IF EDGEPOS(MC_BR_AsmPowerOn_AcpTrak_0.Done)THEN
				CntShuttle := 1;
				VisCappingStates:=1;
				VisPouringStates[0]:=1;
				VisPouringStates[1]:=1;
				IF NOT(Shuttles_exist) THEN
					Step := ADD_SHUTTLE;
				ELSE
					Step := READY;
				END_IF
			END_IF

			// Adding Shuttles for simulation
		ADD_SHUTTLE:
			IF (MC_BR_SecAddShuttle_AcpTrak_0.Done) THEN
				CntShuttle := CntShuttle + 1;

			ELSIF (CntShuttle <= NUM_SIM_SHUTTLES) THEN
				MC_BR_SecAddShuttle_AcpTrak_0.Sector   := ADR(SectorBottleInput);
				MC_BR_SecAddShuttle_AcpTrak_0.Execute  := TRUE;
				MC_BR_SecAddShuttle_AcpTrak_0.Position := SimShuttlePosition[CntShuttle];
				MC_BR_SecAddShuttle_AcpTrak_0.AdvancedParameters.Velocity := 0.0;
			ELSE
				CntShuttle := 1;
				Step := GET_SHUTTLE;
			END_IF

			// Get all availableJadded ones in the simulation
		GET_SHUTTLE:

			MC_BR_AsmGetShuttle_AcpTrak_0.Enable := TRUE;
			IF (MC_BR_AsmGetShuttle_AcpTrak_0.Valid) THEN
				IF (MC_BR_AsmGetShuttle_AcpTrak_0.RemainingCount <> (MC_BR_AsmGetShuttle_AcpTrak_0.TotalCount - CntShuttle)) THEN
					CntShuttle := CntShuttle + 1;
					MC_BR_AsmGetShuttle_AcpTrak_0.Next := FALSE;
				ELSE
					//Save all Axis References to an array for global movement commands*)
					ShuttleAxis[CntShuttle] := MC_BR_AsmGetShuttle_AcpTrak_0.Axis;
					// Get next Shuttle reference with positive Edge on .next
					MC_BR_AsmGetShuttle_AcpTrak_0.Next := TRUE;

					IF (MC_BR_AsmGetShuttle_AcpTrak_0.RemainingCount = 0) THEN
						MC_BR_AsmGetShuttle_AcpTrak_0.Enable := FALSE;
						MC_BR_AsmGetShuttle_AcpTrak_0.Next := FALSE;
						Shuttles_exist := TRUE;
						CntShuttle:=0;
						Step := READY;
					END_IF
				END_IF
			END_IF

			// Active track and ready for command
		READY:
			VisTrakStates:=2;
			// Power off command
			ManualShuttleReset:=0;
			CntShuttle := 1;
			IF (gTrakAsm.Command.Power = FALSE) THEN
				Step := POWER_OFF;
				// Starting main Step - process
			ELSIF VisManual=TRUE THEN
				Step := MANUAL;
			ELSIF (gTrakAsm.Command.ShuttleStart) THEN
				gTrakAsm.Command.ShuttleStart := FALSE;
				VisShuttleStart:=FALSE;
				IF gColorSum=0 THEN
					gColorSum := gOrder.bottlesPerPackage * gOrder.numberOfPackages;
				END_IF;
				IF gColorSum<>0 THEN
					gProcessFinished := FALSE;
					Step := PROCESS;
				ELSE
					NullOrder:=TRUE;
				END_IF;

			ELSIF 	gTrakAsm.Command.ShuttleStop THEN
				Step:=STOPPING;

			END_IF
			IF gPartyOn THEN
				Step:=DELTA_TURN;
				ManualShuttleReset:=0;
			END_IF;
			IF gTrakAsm.Command.Power=FALSE THEN
				Step:=STOPPING;
			END_IF;
			// Main Step, where Shattles run
		PROCESS:

			// if station have no action, its states remain Ready
			IF TON_Pouring_Down.IN THEN
				VisPouringStates[0]:=3;
			ELSE
				VisPouringStates[0]:=2;
			END_IF;
			IF TON_Pouring_Top.IN THEN
				VisPouringStates[1]:=3;
			ELSE
				VisPouringStates[1]:=2;
			END_IF;
			IF TON_Capping.IN THEN
				VisCappingStates:=3;
			ELSE
				VisCappingStates:=2;
			END_IF;
			VisTrakStates:=3;

			FOR ActiveShuttle:=NUM_SIM_SHUTTLES TO 1 BY -1 DO
				MC_BR_ShReadInfo_AcpTrak_0.Enable:=FALSE;
				MC_BR_ShReadInfo_AcpTrak_0();
				MC_BR_ShReadInfo_AcpTrak_0.Axis:= ADR(ShuttleAxis[ActiveShuttle]); //ActiveShuttle
				MC_BR_ShReadInfo_AcpTrak_0.Enable:=TRUE;
				MC_BR_ShReadInfo_AcpTrak_0();
				MC_BR_RoutedMoveAbs_AcpTrak_0.Execute:=FALSE;
				MC_BR_RoutedMoveAbs_AcpTrak_0();

				// States of running shuttles

				IF  MC_BR_ShReadInfo_AcpTrak_0.ShuttleInfo.CurrentValues.SectorName = 'SectorBottleInput' THEN
					Step_Sector:=Bottle_Input;
					IF NOT(Stop_With_Execution) THEN
						gShuttleInPlace_Input:=TRUE;
					END_IF;

					IF gBottleInPlace_Input=TRUE THEN
						BottleVisibility[ActiveShuttle-1]:=TRUE;
						Step_Sector:=WaitPour;
						gBottleInPlace_Input:=FALSE;
						gShuttleInPlace_Input:=FALSE;
					END_IF;

				ELSIF MC_BR_ShReadInfo_AcpTrak_0.ShuttleInfo.RouteDestinationInfo.SectorName = 'SectorBottleInput' THEN
					Step_Sector:=Bottle_Input;

				ELSIF   MC_BR_ShReadInfo_AcpTrak_0.ShuttleInfo.CurrentValues.SectorName = 'SectorWaitPour' THEN
					Step_Sector:=WaitPour;
					// Pouring arrive
					IF Pouring_Down_Comming=FALSE AND Step_Sector=WaitPour  THEN
						Step_Sector:=Pouring_Down;
					END_IF;
					IF Pouring_Down_Comming=TRUE AND Step_Sector=WaitPour AND Pouring_Top_Comming=FALSE  THEN
						Step_Sector:=Pouring_Top;
					END_IF;

				ELSIF  MC_BR_ShReadInfo_AcpTrak_0.ShuttleInfo.RouteDestinationInfo.SectorName = 'SectorWaitPour' THEN
					Step_Sector:=WaitPour;

				ELSIF   MC_BR_ShReadInfo_AcpTrak_0.ShuttleInfo.CurrentValues.SectorName = 'SectorPouring_Down'
					OR MC_BR_ShReadInfo_AcpTrak_0.ShuttleInfo.RouteDestinationInfo.SectorName = 'SectorPouring_Down'
					THEN
					Step_Sector:=Pouring_Down;

					//Pouring done and sending shuttle to capping queue
					IF   TON_Pouring_Down.Q THEN
						Pouring_Down_Busy:=FALSE;
						Pouring_Down_Comming:=FALSE;
						Step_Sector:=WaitCap;
						TON_Pouring_Down.IN:=FALSE;
					END_IF

				ELSIF   MC_BR_ShReadInfo_AcpTrak_0.ShuttleInfo.CurrentValues.SectorName = 'SectorPouring_Top'
					OR MC_BR_ShReadInfo_AcpTrak_0.ShuttleInfo.RouteDestinationInfo.SectorName = 'SectorPouring_Top'
					THEN
					Step_Sector:=Pouring_Top;

					//Pouring done and sending shuttle to capping queue
					IF   TON_Pouring_Top.Q THEN
						Pouring_Top_Busy:=FALSE;
						Pouring_Top_Comming:=FALSE;
						Step_Sector:=WaitCap;
						TON_Pouring_Top.IN:=FALSE;
					END_IF

				ELSIF   MC_BR_ShReadInfo_AcpTrak_0.ShuttleInfo.CurrentValues.SectorName = 'SectorWaitCapping' THEN
					Step_Sector:=WaitCap;

					// Sending shuttle to capping if its idle
					IF Step_Sector=WaitCap AND Capping_Comming=FALSE AND Capping_Broken = FALSE THEN
						Step_Sector:=Capping;
					END_IF;
				ELSIF  MC_BR_ShReadInfo_AcpTrak_0.ShuttleInfo.RouteDestinationInfo.SectorName = 'SectorWaitCapping' THEN
					Step_Sector:=WaitCap;

				ELSIF   MC_BR_ShReadInfo_AcpTrak_0.ShuttleInfo.CurrentValues.SectorName = 'SectorCapping'
					OR MC_BR_ShReadInfo_AcpTrak_0.ShuttleInfo.RouteDestinationInfo.SectorName = 'SectorCapping'
					THEN
					Step_Sector:=Capping;

					// After capping sendig to delivery
					IF  TON_Capping.Q THEN
						Capping_Busy := FALSE;
						Step_Sector:=Bottle_Output;
						TON_Capping.IN:=FALSE;
						Capping_Comming:=FALSE;
					END_IF
				ELSIF   MC_BR_ShReadInfo_AcpTrak_0.ShuttleInfo.CurrentValues.SectorName = 'SectorBottleOutput' THEN
					Step_Sector:=Bottle_Output;
					gShuttleInPlace_Output:=TRUE;

					// bottle in place for delivery waiting for signal and then sending shuttle to sector input
					IF gBottleInPlace_Output=TRUE THEN
						BottleVisibility[ActiveShuttle-1]:=FALSE;
						BottleMaterial[ActiveShuttle-1]:=13;
						Step_Sector:=Bottle_Input;
						gBottleInPlace_Output:=FALSE;
						gShuttleInPlace_Output:=FALSE;
					END_IF;

				ELSIF MC_BR_ShReadInfo_AcpTrak_0.ShuttleInfo.RouteDestinationInfo.SectorName = 'SectorBottleOutput' THEN
					Step_Sector:=Bottle_Output;
				END_IF;

				// TON activation
				IF Pouring_Top_Busy=TRUE THEN
					TON_Pouring_Top.IN:=TRUE;
				END_IF;
				IF Pouring_Down_Busy=TRUE THEN
					TON_Pouring_Down.IN:=TRUE;
				END_IF;
				IF Capping_Busy=TRUE THEN
					TON_Capping.IN:=TRUE;
				END_IF;
				//Handling broken stations
				IF Pouring_Down_Broken THEN
					VisPouringStates[0]:=4;
					Pouring_Down_Comming:=TRUE;
					SvgTranform[3]:=2;
				END_IF
				IF EDGENEG(Pouring_Down_Broken) THEN
					Pouring_Down_Comming:=FALSE;
					SvgTranform[3]:=0;
				END_IF;
				IF Pouring_Top_Broken THEN
					VisPouringStates[1]:=4;
					Pouring_Top_Comming:=TRUE;
					SvgTranform[4]:=2;
				END_IF;
				IF EDGENEG(Pouring_Top_Broken) THEN
					Pouring_Top_Comming:=FALSE;
					SvgTranform[4]:=0;
				END_IF;
				IF Capping_Broken THEN
					VisCappingStates:=4;
					Capping_Comming:=TRUE;
					SvgTranform[2]:=2;
				END_IF

				// Step for active Shuttle
				CASE Step_Sector OF

					// Bottle input at Shuttel
					Bottle_Input:
						gShuttleColored[NUM_SIM_SHUTTLES-ActiveShuttle]:=FALSE;
						gShuttleColor[NUM_SIM_SHUTTLES-ActiveShuttle] := 0;
						MC_BR_RoutedMoveAbs_AcpTrak_0.Axis          := ADR(ShuttleAxis[ActiveShuttle]);
						MC_BR_RoutedMoveAbs_AcpTrak_0.Execute       := TRUE;
						MC_BR_RoutedMoveAbs_AcpTrak_0.Sector        := ADR(SectorBottleInput);
						MC_BR_RoutedMoveAbs_AcpTrak_0.Position      := 0.305+3.66;
						// Wait for pouring if Pouring_A/_B are busy
					WaitPour:
						MC_BR_RoutedMoveAbs_AcpTrak_0.Axis          := ADR(ShuttleAxis[ActiveShuttle]);
						MC_BR_RoutedMoveAbs_AcpTrak_0.Execute       := TRUE;
						MC_BR_RoutedMoveAbs_AcpTrak_0.Sector        := ADR(SectorWaitPour);
						MC_BR_RoutedMoveAbs_AcpTrak_0.Position      := 0.6;

						// Pouring bottle in down station
					Pouring_Down:
						Pouring_Down_Comming:=TRUE;
						IF  MC_BR_ShReadInfo_AcpTrak_0.ShuttleInfo.CurrentValues.SectorName = 'SectorPouring_Down' THEN
							Pouring_Down_Busy:=TRUE;
							IF NOT (gShuttleColored[NUM_SIM_SHUTTLES-ActiveShuttle]) THEN
								CASE gOrder.drinkColor OF
									DRINK_COLOR_RED:
										BottleMaterial[ActiveShuttle-1]:=1;
										gShuttleColor[NUM_SIM_SHUTTLES-ActiveShuttle] := 2;
										gShuttleColored[NUM_SIM_SHUTTLES-ActiveShuttle] := TRUE;
									DRINK_COLOR_GREEN:
										BottleMaterial[ActiveShuttle-1]:=5;
										gShuttleColor[NUM_SIM_SHUTTLES-ActiveShuttle] := 1;
										gShuttleColored[NUM_SIM_SHUTTLES-ActiveShuttle] := TRUE;
									DRINK_COLOR_BLUE:
										BottleMaterial[ActiveShuttle-1]:=2;
										gShuttleColor[NUM_SIM_SHUTTLES-ActiveShuttle] := 3;
										gShuttleColored[NUM_SIM_SHUTTLES-ActiveShuttle] := TRUE;
								END_CASE;
							END_IF;
						END_IF;
						MC_BR_RoutedMoveAbs_AcpTrak_0.Axis          := ADR(ShuttleAxis[ActiveShuttle]);
						MC_BR_RoutedMoveAbs_AcpTrak_0.Execute       := TRUE;
						MC_BR_RoutedMoveAbs_AcpTrak_0.Sector        := ADR(SectorPouring_Down);
						CASE gOrder.drinkColor OF
							DRINK_COLOR_RED:
								MC_BR_RoutedMoveAbs_AcpTrak_0.Position      := 0.05;
							DRINK_COLOR_GREEN:
								MC_BR_RoutedMoveAbs_AcpTrak_0.Position      := 0.20;
							DRINK_COLOR_BLUE:
								MC_BR_RoutedMoveAbs_AcpTrak_0.Position      := 0.35;
						END_CASE;
						// Pouring bottle in Top station
					Pouring_Top:
						Pouring_Top_Comming   :=TRUE;
						IF  MC_BR_ShReadInfo_AcpTrak_0.ShuttleInfo.CurrentValues.SectorName = 'SectorPouring_Top' THEN
							Pouring_Top_Busy := TRUE;
							IF NOT (gShuttleColored[NUM_SIM_SHUTTLES-ActiveShuttle]) THEN
								CASE gOrder.drinkColor OF
									DRINK_COLOR_RED:
										BottleMaterial[ActiveShuttle-1]:=1;
										gShuttleColor[NUM_SIM_SHUTTLES-ActiveShuttle] := 2;
										gShuttleColored[NUM_SIM_SHUTTLES-ActiveShuttle] := TRUE;
									DRINK_COLOR_GREEN:
										BottleMaterial[ActiveShuttle-1]:=5;
										gShuttleColor[NUM_SIM_SHUTTLES-ActiveShuttle] := 1;
										gShuttleColored[NUM_SIM_SHUTTLES-ActiveShuttle] := TRUE;
									DRINK_COLOR_BLUE:
										BottleMaterial[ActiveShuttle-1]:=2;
										gShuttleColor[NUM_SIM_SHUTTLES-ActiveShuttle] := 3;
										gShuttleColored[NUM_SIM_SHUTTLES-ActiveShuttle] := TRUE;
								END_CASE;
							END_IF;
						END_IF;
						MC_BR_RoutedMoveAbs_AcpTrak_0.Axis          := ADR(ShuttleAxis[ActiveShuttle]);
						MC_BR_RoutedMoveAbs_AcpTrak_0.Execute       := TRUE;
						MC_BR_RoutedMoveAbs_AcpTrak_0.Sector        := ADR(SectorPouring_Top);
						CASE gOrder.drinkColor OF
							DRINK_COLOR_RED:
								MC_BR_RoutedMoveAbs_AcpTrak_0.Position      := 0.05;
							DRINK_COLOR_GREEN:
								MC_BR_RoutedMoveAbs_AcpTrak_0.Position      := 0.20;
							DRINK_COLOR_BLUE:
								MC_BR_RoutedMoveAbs_AcpTrak_0.Position      := 0.35;
						END_CASE;

						// Wait for capping if Cap station is busy
					WaitCap:
						MC_BR_RoutedMoveAbs_AcpTrak_0.Axis          := ADR(ShuttleAxis[ActiveShuttle]);
						MC_BR_RoutedMoveAbs_AcpTrak_0.Execute       := TRUE;
						MC_BR_RoutedMoveAbs_AcpTrak_0.Sector        := ADR(SectorWaitCapping);
						MC_BR_RoutedMoveAbs_AcpTrak_0.Position      := 0.5;

						// Capping a bottle
					Capping:
						Capping_Comming  := TRUE;
						IF  MC_BR_ShReadInfo_AcpTrak_0.ShuttleInfo.CurrentValues.SectorName = 'SectorCapping' THEN
							Capping_Busy := TRUE;
						END_IF;
						MC_BR_RoutedMoveAbs_AcpTrak_0.Axis          := ADR(ShuttleAxis[ActiveShuttle]);
						MC_BR_RoutedMoveAbs_AcpTrak_0.Execute       := TRUE;
						MC_BR_RoutedMoveAbs_AcpTrak_0.Sector        := ADR(SectorCapping);
						MC_BR_RoutedMoveAbs_AcpTrak_0.Position      := 0.305;

						// Take bottle from Shuttel
					Bottle_Output:
						MC_BR_RoutedMoveAbs_AcpTrak_0.Axis          := ADR(ShuttleAxis[ActiveShuttle]);
						MC_BR_RoutedMoveAbs_AcpTrak_0.Execute       := TRUE;
						MC_BR_RoutedMoveAbs_AcpTrak_0.Sector        := ADR(SectorBottleOutput);
						MC_BR_RoutedMoveAbs_AcpTrak_0.Position      := 0.305;
				END_CASE;

				MC_BR_RoutedMoveAbs_AcpTrak_0.Velocity      := gTrakAsm.Parameter.Velocity;
				MC_BR_RoutedMoveAbs_AcpTrak_0.Acceleration  := gTrakAsm.Parameter.Acceleration;
				MC_BR_RoutedMoveAbs_AcpTrak_0.Deceleration  := gTrakAsm.Parameter.Deceleration;
				MC_BR_RoutedMoveAbs_AcpTrak_0.Jerk          := 0.0;
				MC_BR_RoutedMoveAbs_AcpTrak_0.BufferMode    := mcABORTING;
				MC_BR_RoutedMoveAbs_AcpTrak_0.AdvancedParameters.StartDirection     := mcDIR_UNDEFINED;
				MC_BR_RoutedMoveAbs_AcpTrak_0.AdvancedParameters.EndDirection       := mcDIR_POSITIVE;
				MC_BR_RoutedMoveAbs_AcpTrak_0.AdvancedParameters.ShuttleOrientation := mcDIR_UNDEFINED;
				MC_BR_RoutedMoveAbs_AcpTrak_0();

				IF MC_BR_ShReadInfo_AcpTrak_0.ShuttleInfo.RouteDestinationInfo.RemainingDistance < 1
					AND gColorSum=0 AND (MC_BR_ShReadInfo_AcpTrak_0.ShuttleInfo.CurrentValues.SectorName='SectorBottleInput' OR
					MC_BR_ShReadInfo_AcpTrak_0.ShuttleInfo.RouteDestinationInfo.SectorName='SectorBottleInput') THEN
					ManualShuttleReset:= ManualShuttleReset +1;
				END_IF;
			END_FOR;

			IF Capping_Busy THEN
				IF Capping_Position=350 THEN
					Capping_Rotate:=Capping_Rotate+24;
					IF Capping_Rotate=360 THEN
						Capping_Rotate:=0;
					END_IF;
				ELSE
					Capping_Position:=Capping_Position-5;
				END_IF;
			ELSE
				IF NOT(Capping_Position=450) THEN
					Capping_Position:=Capping_Position+5;
				END_IF;
			END_IF;
			IF Pouring_Top_Busy THEN
				IF NOT (Pouring_Top_Position=350) THEN
					Pouring_Top_Position:=Pouring_Top_Position-5;
				END_IF;
			ELSE
				IF NOT (Pouring_Top_Position=400) THEN
					Pouring_Top_Position:=Pouring_Top_Position+5;
				END_IF;
			END_IF;
			IF Pouring_Down_Busy THEN
				IF NOT (Pouring_Down_Position=350) THEN
					Pouring_Down_Position:=Pouring_Down_Position-5;
				END_IF;
			ELSE
				IF NOT (Pouring_Down_Position=400) THEN
					Pouring_Down_Position:=Pouring_Down_Position+5;
				END_IF;
			END_IF;
			IF Stop_With_Execution THEN
				ManualShuttleReset:=0;
				FOR ActiveShuttle:=NUM_SIM_SHUTTLES TO 1 BY -1 DO
					MC_BR_ShReadInfo_AcpTrak_0.Enable:=FALSE;
					MC_BR_ShReadInfo_AcpTrak_0();
					MC_BR_ShReadInfo_AcpTrak_0.Axis:= ADR(ShuttleAxis[ActiveShuttle]); //ActiveShuttle
					MC_BR_ShReadInfo_AcpTrak_0.Enable:=TRUE;
					MC_BR_ShReadInfo_AcpTrak_0();

					IF MC_BR_ShReadInfo_AcpTrak_0.ShuttleInfo.RouteDestinationInfo.RemainingDistance < 1
						AND (MC_BR_ShReadInfo_AcpTrak_0.ShuttleInfo.CurrentValues.SectorName='SectorBottleInput' OR
						MC_BR_ShReadInfo_AcpTrak_0.ShuttleInfo.RouteDestinationInfo.SectorName='SectorBottleInput') THEN
						ManualShuttleReset:= ManualShuttleReset +1;
					END_IF;
				END_FOR;
			END_IF;
			IF ManualShuttleReset=NUM_SIM_SHUTTLES THEN
				Step:=READY;
				gProcessFinished := TRUE;
				VisShuttleStart:=FALSE;
				Stop_With_Execution:=FALSE;
			ELSE
				ManualShuttleReset:=0;
			END_IF

			// Stop command
			IF(gTrakAsm.Command.ShuttleStop) OR VisManual=TRUE THEN
				CntShuttle := 1;
				Step := STOPPING;
			END_IF

			// Error stop
			IF (MC_BR_RoutedMoveVel_AcpTrak_0.Error) THEN
				MC_BR_AsmReset_AcpTrak_0.Execute := TRUE;
				Step := RESET;
			END_IF
			IF gPartyOn THEN
				Step:=DELTA_TURN;
				ManualShuttleReset:=0;
			END_IF;
			// Machine States
			IF gTrakAsm.Command.Power=FALSE THEN
				Step:=STOPPING;
			END_IF;

		MANUAL:
			VisTrakStates:=5;
			IF VisManual=FALSE THEN

				FOR CntShuttle:=NUM_SIM_SHUTTLES TO 1 BY -1 DO
					MC_BR_RoutedMoveAbs_AcpTrak_0.Execute:=FALSE;
					MC_BR_RoutedMoveAbs_AcpTrak_0();
					MC_BR_RoutedMoveAbs_AcpTrak_0.Axis         							:= ADR(ShuttleAxis[CntShuttle]);
					MC_BR_RoutedMoveAbs_AcpTrak_0.Execute      						 	:= TRUE;
					MC_BR_RoutedMoveAbs_AcpTrak_0.Sector       					 		:= ADR(SectorBottleInput);
					MC_BR_RoutedMoveAbs_AcpTrak_0.Position     						    := 0.305+3.66;
					MC_BR_RoutedMoveAbs_AcpTrak_0.Velocity      						:= gTrakAsm.Parameter.Velocity;
					MC_BR_RoutedMoveAbs_AcpTrak_0.Acceleration  						:= gTrakAsm.Parameter.Acceleration;
					MC_BR_RoutedMoveAbs_AcpTrak_0.Deceleration  						:= gTrakAsm.Parameter.Deceleration;
					MC_BR_RoutedMoveAbs_AcpTrak_0.Jerk          						:= 0.0;
					MC_BR_RoutedMoveAbs_AcpTrak_0.BufferMode    						:= mcABORTING;
					MC_BR_RoutedMoveAbs_AcpTrak_0.AdvancedParameters.StartDirection     := mcDIR_UNDEFINED;
					MC_BR_RoutedMoveAbs_AcpTrak_0.AdvancedParameters.EndDirection       := mcDIR_POSITIVE;
					MC_BR_RoutedMoveAbs_AcpTrak_0.AdvancedParameters.ShuttleOrientation := mcDIR_UNDEFINED;
					MC_BR_RoutedMoveAbs_AcpTrak_0();
					MC_BR_ShReadInfo_AcpTrak_0.Enable									:=FALSE;
					MC_BR_ShReadInfo_AcpTrak_0();
					MC_BR_ShReadInfo_AcpTrak_0.Axis 									:=ADR(ShuttleAxis[CntShuttle]);
					MC_BR_ShReadInfo_AcpTrak_0.Enable									:=TRUE;
					MC_BR_ShReadInfo_AcpTrak_0();
					IF MC_BR_ShReadInfo_AcpTrak_0.ShuttleInfo.RouteDestinationInfo.RemainingDistance < 1.5
						AND  (MC_BR_ShReadInfo_AcpTrak_0.ShuttleInfo.CurrentValues.SectorName='SectorBottleInput' OR
						MC_BR_ShReadInfo_AcpTrak_0.ShuttleInfo.RouteDestinationInfo.SectorName='SectorBottleInput') THEN
						ManualShuttleReset:= ManualShuttleReset +1;
					END_IF;
				END_FOR;
				IF Pouring_Down_Position<>400 THEN
					IF Pouring_Down_Position<400 THEN
						Pouring_Down_Position:=Pouring_Down_Position+5;
					END_IF;
					IF Pouring_Down_Position>400 THEN
						Pouring_Down_Position:=Pouring_Down_Position-5;
					END_IF;
				END_IF;
				IF Pouring_Top_Position<>400 THEN
					IF Pouring_Top_Position<400 THEN
						Pouring_Top_Position:=Pouring_Top_Position+5;
					END_IF;
					IF Pouring_Down_Position>400 THEN
						Pouring_Top_Position:=Pouring_Top_Position-5;
					END_IF;
				END_IF;
				IF Capping_Position<>400 THEN
					IF Capping_Position<400 THEN
						Capping_Position:=Capping_Position+5;
					END_IF;
					IF Capping_Position>400 THEN
						Capping_Position:=Capping_Position-5;
					END_IF;
				END_IF;
				IF Capping_Rotate<>0 THEN
					Capping_Rotate:=Capping_Rotate-12;
				END_IF;
				IF ManualShuttleReset=NUM_SIM_SHUTTLES AND Capping_Position=400 AND Pouring_Top_Position=400 AND Pouring_Down_Position=400 THEN
					CntShuttle:=1;
					Step := READY;
					Pouring_Top_Comming:=FALSE;
					Pouring_Down_Comming:=FALSE;
					Pouring_Top_Busy:=FALSE;
					Pouring_Down_Busy:=FALSE;
					Capping_Comming:=FALSE;
					Capping_Busy:=FALSE;
					gShuttleInPlace_Input:=FALSE;
					gShuttleInPlace_Output:=FALSE;
					TON_Pouring_Down.IN:=FALSE;
					TON_Pouring_Top.IN:=FALSE;

				END_IF;
			ELSE 		// MANUAL TURNED ON
				IF VisCappingRotate THEN
					Capping_Rotate:=Capping_Rotate+12;
					IF Capping_Rotate=360 THEN
						Capping_Rotate:=0;
					END_IF;
				END_IF;
				IF VisCappingAdd AND Capping_Position<500 THEN
					Capping_Position:= Capping_Position+5;
				END_IF;
				IF VisCappingSub AND Capping_Position>200 THEN
					Capping_Position:= Capping_Position-5;
				END_IF;
				IF VisPouringNumber =0 THEN
					IF VisPouringAdd AND Pouring_Top_Position<450 THEN
						Pouring_Top_Position:=Pouring_Top_Position+5;
					END_IF;
					IF VisPouringSub AND Pouring_Top_Position>200 THEN
						Pouring_Top_Position:=Pouring_Top_Position-5;
					END_IF;
				ELSIF VisPouringNumber = 1 THEN
					IF VisPouringAdd AND Pouring_Down_Position<450 THEN
						Pouring_Down_Position:=Pouring_Down_Position+5;
					END_IF;
					IF VisPouringSub AND Pouring_Down_Position>200 THEN
						Pouring_Down_Position:=Pouring_Down_Position-5;
					END_IF;
				END_IF;

				MC_BR_RoutedMoveVel_AcpTrak_0.Execute		:=FALSE;
				MC_BR_RoutedMoveVel_AcpTrak_0();
				MC_BR_RoutedMoveVel_AcpTrak_0.Axis			:=ADR(ShuttleAxis[VisShuttle+1]);
				MC_BR_RoutedMoveVel_AcpTrak_0.Execute		:=TRUE;
				IF VisManualSectorTop=TRUE THEN
					MC_BR_RoutedMoveVel_AcpTrak_0.Sector        := ADR(SectorManualTop);
				ELSE
					MC_BR_RoutedMoveVel_AcpTrak_0.Sector        := ADR(SectorManualMain);
				END_IF;
				IF VisMove_Pos THEN
					MC_BR_RoutedMoveVel_AcpTrak_0.Velocity      := VisManualVelocity;
				ELSIF VisMove_Neg THEN
					MC_BR_RoutedMoveVel_AcpTrak_0.Velocity      := VisManualVelocity;
				ELSE
					MC_BR_RoutedMoveVel_AcpTrak_0.Velocity  := 0.0;
				END_IF;
				MC_BR_RoutedMoveVel_AcpTrak_0.Acceleration  := gTrakAsm.Parameter.Acceleration;
				MC_BR_RoutedMoveVel_AcpTrak_0.Deceleration  := gTrakAsm.Parameter.Deceleration;
				MC_BR_RoutedMoveVel_AcpTrak_0.Jerk          := 0.0;
				MC_BR_RoutedMoveVel_AcpTrak_0.BufferMode    := mcABORTING;
				IF VisMove_Pos THEN
					MC_BR_RoutedMoveVel_AcpTrak_0.AdvancedParameters.EndDirection       := mcDIR_POSITIVE;
				ELSE
					MC_BR_RoutedMoveVel_AcpTrak_0.AdvancedParameters.EndDirection       := mcDIR_NEGATIVE;
				END_IF;
				MC_BR_RoutedMoveVel_AcpTrak_0.AdvancedParameters.ShuttleOrientation := mcDIR_UNDEFINED;

				MC_BR_RoutedMoveVel_AcpTrak_0.AdvancedParameters.StartDirection     := mcDIR_UNDEFINED;
			END_IF
			ManualShuttleReset:=0;

			IF gPartyOn THEN
				Step:=DELTA_TURN;
				ManualShuttleReset:=0;
			END_IF;
			IF gTrakAsm.Command.Power=FALSE THEN
	  			Step:=STOPPING;
			END_IF;

		STOPPING:
			VisTrakStates:=4;
			gShuttleInPlace_Input:=FALSE;
			gShuttleInPlace_Output:=FALSE;
			gShuttleInPlace_Turn:=FALSE;
			FOR CntShuttle:=NUM_SIM_SHUTTLES TO 1 BY -1 DO
				MC_BR_ShReadInfo_AcpTrak_0.Enable									:=FALSE;
				MC_BR_ShReadInfo_AcpTrak_0();
				MC_BR_ShReadInfo_AcpTrak_0.Axis 									:=ADR(ShuttleAxis[CntShuttle]);
				MC_BR_ShReadInfo_AcpTrak_0.Enable									:=TRUE;
				MC_BR_ShReadInfo_AcpTrak_0();
				MC_BR_RoutedMoveVel_AcpTrak_0.Execute:=FALSE;
				MC_BR_RoutedMoveVel_AcpTrak_0();
				MC_BR_RoutedMoveVel_AcpTrak_0.Axis         							:= ADR(ShuttleAxis[CntShuttle]);
				MC_BR_RoutedMoveVel_AcpTrak_0.Execute      						 	:= TRUE;
				IF MC_BR_ShReadInfo_AcpTrak_0.ShuttleInfo.CurrentValues.SectorName='SectorBottleInput'
					OR MC_BR_ShReadInfo_AcpTrak_0.ShuttleInfo.RouteDestinationInfo.SectorName='SectorBottleInput'
					THEN
					MC_BR_RoutedMoveVel_AcpTrak_0.Sector       					 		:= ADR(SectorBottleInput);
				ELSIF MC_BR_ShReadInfo_AcpTrak_0.ShuttleInfo.CurrentValues.SectorName='SectorBottleOutput'
					OR MC_BR_ShReadInfo_AcpTrak_0.ShuttleInfo.RouteDestinationInfo.SectorName='SectorBottleOutput'
					THEN
					MC_BR_RoutedMoveVel_AcpTrak_0.Sector       					 		:= ADR(SectorBottleOutput);
				ELSIF MC_BR_ShReadInfo_AcpTrak_0.ShuttleInfo.CurrentValues.SectorName='SectorWaitPour'
					OR MC_BR_ShReadInfo_AcpTrak_0.ShuttleInfo.RouteDestinationInfo.SectorName='SectorWaitPour'
					THEN
					MC_BR_RoutedMoveVel_AcpTrak_0.Sector       					 		:= ADR(SectorWaitPour);
				ELSIF MC_BR_ShReadInfo_AcpTrak_0.ShuttleInfo.CurrentValues.SectorName='SectorPouring_Down'
					OR MC_BR_ShReadInfo_AcpTrak_0.ShuttleInfo.RouteDestinationInfo.SectorName='SectorPouring_Down'
					THEN
					MC_BR_RoutedMoveVel_AcpTrak_0.Sector       					 		:= ADR(SectorPouring_Down);
				ELSIF MC_BR_ShReadInfo_AcpTrak_0.ShuttleInfo.CurrentValues.SectorName='SectorPouring_Top'
					OR MC_BR_ShReadInfo_AcpTrak_0.ShuttleInfo.RouteDestinationInfo.SectorName='SectorPouring_Top'
					THEN
					MC_BR_RoutedMoveVel_AcpTrak_0.Sector       					 		:= ADR(SectorPouring_Top);
				ELSIF MC_BR_ShReadInfo_AcpTrak_0.ShuttleInfo.CurrentValues.SectorName='SectorWaitCapping'
					OR MC_BR_ShReadInfo_AcpTrak_0.ShuttleInfo.RouteDestinationInfo.SectorName='SectorWaitCapping'
					THEN
					MC_BR_RoutedMoveVel_AcpTrak_0.Sector       					 		:= ADR(SectorWaitCapping);
				ELSIF MC_BR_ShReadInfo_AcpTrak_0.ShuttleInfo.CurrentValues.SectorName='SectorCapping'
					OR MC_BR_ShReadInfo_AcpTrak_0.ShuttleInfo.RouteDestinationInfo.SectorName='SectorCapping'
					THEN
					MC_BR_RoutedMoveVel_AcpTrak_0.Sector       					 		:= ADR(SectorCapping);
				END_IF;
				MC_BR_RoutedMoveVel_AcpTrak_0.Position     						    := 0.0;
				MC_BR_RoutedMoveVel_AcpTrak_0.Velocity      						:= 0.0;
				MC_BR_RoutedMoveVel_AcpTrak_0.Acceleration  						:= 35.0;
				MC_BR_RoutedMoveVel_AcpTrak_0.Deceleration  						:= 35.0;
				MC_BR_RoutedMoveVel_AcpTrak_0.Jerk          						:= 0.0;
				MC_BR_RoutedMoveVel_AcpTrak_0.BufferMode    						:= mcABORTING;
				MC_BR_RoutedMoveVel_AcpTrak_0.AdvancedParameters.StartDirection     := mcDIR_UNDEFINED;
				MC_BR_RoutedMoveVel_AcpTrak_0.AdvancedParameters.EndDirection       := mcDIR_POSITIVE;
				MC_BR_RoutedMoveVel_AcpTrak_0.AdvancedParameters.ShuttleOrientation := mcDIR_UNDEFINED;
				MC_BR_RoutedMoveVel_AcpTrak_0();
			END_FOR;
			VisShuttleStop:=FALSE;
			VisShuttleStart:=FALSE;
			Pouring_Top_Comming				:=FALSE;
			Pouring_Down_Comming			:=FALSE;
			Pouring_Top_Busy				:=FALSE;
			Pouring_Down_Busy				:=FALSE;
			Capping_Comming					:=FALSE;
			Capping_Busy					:=FALSE;
			gShuttleInPlace_Input			:=FALSE;
			gShuttleInPlace_Output			:=FALSE;
			TON_Pouring_Down.IN				:=FALSE;
			TON_Pouring_Top.IN				:=FALSE;
			IF VisManual=TRUE THEN
				Step:=MANUAL;
			ELSE
				Step := READY;
			END_IF;
			IF gTrakAsm.Command.Power=FALSE THEN
				Step:=STOPPING;
			END_IF;
			// Reset due to error
		RESET:
			IF EDGEPOS(MC_BR_AsmReset_AcpTrak_0.Done) THEN
				gTrakAsm.Command.ShuttleStart    := FALSE;
				gTrakAsm.Command.ShuttleStop     := FALSE;
				MC_BR_AsmReset_AcpTrak_0.Execute := FALSE;
				MC_BR_RoutedMoveVel_AcpTrak_0.Execute := FALSE;
				Step := READY;
			END_IF

		DELTA_TURN:
			IF DeltaInit=TRUE THEN

			ELSE
				IF ManualShuttleReset=NUM_SIM_SHUTTLES THEN
					FOR DeltaFor:=NUM_SIM_SHUTTLES TO 1 BY -1 DO
						MC_BR_RoutedMoveAbs_AcpTrak_0.Execute								:=FALSE;
						MC_BR_RoutedMoveAbs_AcpTrak_0();
						MC_BR_RoutedMoveAbs_AcpTrak_0.Axis         							:= ADR(ShuttleAxis[DeltaFor]);
						MC_BR_RoutedMoveAbs_AcpTrak_0.Sector       					 		:= ADR(SectorManualTop);
						MC_BR_RoutedMoveAbs_AcpTrak_0.Execute								:= TRUE;
						MC_BR_RoutedMoveAbs_AcpTrak_0.Position     						    := 1.4*DeltaFor;
						MC_BR_RoutedMoveAbs_AcpTrak_0.Velocity      						:= 1.0;
						MC_BR_RoutedMoveAbs_AcpTrak_0.Acceleration  						:= 5.0;
						MC_BR_RoutedMoveAbs_AcpTrak_0.Deceleration  						:= 5.0;
						MC_BR_RoutedMoveAbs_AcpTrak_0.Jerk          						:= 0.0;
						MC_BR_RoutedMoveAbs_AcpTrak_0.BufferMode    						:= mcABORTING;
						MC_BR_RoutedMoveAbs_AcpTrak_0.AdvancedParameters.StartDirection     := mcDIR_UNDEFINED;
						IF DeltaFor>8 THEN
							MC_BR_RoutedMoveAbs_AcpTrak_0.AdvancedParameters.EndDirection       := mcDIR_POSITIVE;
						ELSE
							MC_BR_RoutedMoveAbs_AcpTrak_0.AdvancedParameters.EndDirection       := mcDIR_NEGATIVE;
						END_IF;
						MC_BR_RoutedMoveAbs_AcpTrak_0.AdvancedParameters.ShuttleOrientation := mcDIR_UNDEFINED;
						IF TON_Delta.Q=FALSE THEN
							MC_BR_RoutedMoveAbs_AcpTrak_0();
						END_IF;
						gShuttleColor[DeltaFor] := 3;
						IF gShuttleColor[DeltaFor-1]=3 THEN
							gShuttleColor[DeltaFor] := 1;
						ELSE
							gShuttleColor[DeltaFor] := 3;
						END_IF;
					END_FOR;
					TON_Delta.IN:=TRUE;
					Step:=DELTA_MOVE;
				ELSE
					ManualShuttleReset:=0;
					FOR DeltaFor:=NUM_SIM_SHUTTLES TO 1 BY -1 DO
						MC_BR_RoutedMoveAbs_AcpTrak_0.Execute								:=FALSE;
						MC_BR_RoutedMoveAbs_AcpTrak_0();
						MC_BR_RoutedMoveAbs_AcpTrak_0.Axis         							:= ADR(ShuttleAxis[DeltaFor]);
						MC_BR_RoutedMoveAbs_AcpTrak_0.Execute      						 	:= TRUE;
						MC_BR_RoutedMoveAbs_AcpTrak_0.Sector       					 		:= ADR(SectorWaitPour);
						MC_BR_RoutedMoveAbs_AcpTrak_0.Position     						    := 0.5;
						MC_BR_RoutedMoveAbs_AcpTrak_0.Velocity      						:= 4;
						MC_BR_RoutedMoveAbs_AcpTrak_0.Acceleration  						:= 40.0;
						MC_BR_RoutedMoveAbs_AcpTrak_0.Deceleration  						:= 40.0;
						MC_BR_RoutedMoveAbs_AcpTrak_0.Jerk          						:= 0.0;
						MC_BR_RoutedMoveAbs_AcpTrak_0.BufferMode    						:= mcABORTING;
						MC_BR_RoutedMoveAbs_AcpTrak_0.AdvancedParameters.StartDirection     := mcDIR_UNDEFINED;
						MC_BR_RoutedMoveAbs_AcpTrak_0.AdvancedParameters.EndDirection       := mcDIR_POSITIVE;
						MC_BR_RoutedMoveAbs_AcpTrak_0.AdvancedParameters.ShuttleOrientation := mcDIR_UNDEFINED;
						MC_BR_RoutedMoveAbs_AcpTrak_0();
						MC_BR_ShReadInfo_AcpTrak_0.Enable									:=FALSE;
						MC_BR_ShReadInfo_AcpTrak_0();
						MC_BR_ShReadInfo_AcpTrak_0.Axis 									:=ADR(ShuttleAxis[DeltaFor]);
						MC_BR_ShReadInfo_AcpTrak_0.Enable									:=TRUE;
						MC_BR_ShReadInfo_AcpTrak_0();
						IF MC_BR_ShReadInfo_AcpTrak_0.ShuttleInfo.RouteDestinationInfo.RemainingDistance < 0.7
							AND (MC_BR_ShReadInfo_AcpTrak_0.ShuttleInfo.CurrentValues.SectorName='SectorWaitPour' OR
							MC_BR_ShReadInfo_AcpTrak_0.ShuttleInfo.RouteDestinationInfo.SectorName='SectorWaitPour') THEN
							ManualShuttleReset:= ManualShuttleReset +1;
						END_IF;
					END_FOR;
				END_IF;

			END_IF;
			// Stop command
			IF(gTrakAsm.Command.ShuttleStop) OR VisManual=TRUE THEN
				CntShuttle := 1;
				Step := STOPPING;
			END_IF

			// Error stop
			IF (MC_BR_RoutedMoveVel_AcpTrak_0.Error) THEN
				MC_BR_AsmReset_AcpTrak_0.Execute := TRUE;
				Step := RESET;
			END_IF
			IF NOT(gPartyOn) THEN
				Step:=MANUAL;
			END_IF;
			gVisPower:=TRUE;

		DELTA_MOVE:
			IF TON_Delta.Q THEN
				//		DeltaInit:=TRUE;
				FOR DeltaFor:=NUM_SIM_SHUTTLES TO 1 BY -1 DO
					MC_BR_RoutedMoveVel_AcpTrak_0.Execute								:=FALSE;
					MC_BR_RoutedMoveVel_AcpTrak_0();
					MC_BR_RoutedMoveVel_AcpTrak_0.Axis         							:= ADR(ShuttleAxis[DeltaFor]);
					MC_BR_RoutedMoveVel_AcpTrak_0.Sector       					 		:= ADR(SectorManualTop);
					MC_BR_RoutedMoveVel_AcpTrak_0.Execute								:= TRUE;
					MC_BR_RoutedMoveVel_AcpTrak_0.Position     						    := 0.0;
					MC_BR_RoutedMoveVel_AcpTrak_0.Velocity      						:= 4.0;
					MC_BR_RoutedMoveVel_AcpTrak_0.Acceleration  						:= 0.1;
					MC_BR_RoutedMoveVel_AcpTrak_0.Deceleration  						:= gTrakAsm.Parameter.Deceleration;
					MC_BR_RoutedMoveVel_AcpTrak_0.Jerk          						:= 0.0;
					MC_BR_RoutedMoveVel_AcpTrak_0.BufferMode    						:= mcABORTING;
					MC_BR_RoutedMoveVel_AcpTrak_0.AdvancedParameters.StartDirection     := mcDIR_UNDEFINED;
					MC_BR_RoutedMoveVel_AcpTrak_0.AdvancedParameters.EndDirection       := mcDIR_NEGATIVE;
					MC_BR_RoutedMoveVel_AcpTrak_0.AdvancedParameters.ShuttleOrientation := mcDIR_UNDEFINED;
					MC_BR_RoutedMoveVel_AcpTrak_0();
				END_FOR;
				IF gShuttleColor[Delta_Shuttle]=3 THEN
					gShuttleColor[Delta_Shuttle] := 1;
				ELSE
					gShuttleColor[Delta_Shuttle] := 3;
				END_IF;
				Delta_Shuttle:=Delta_Shuttle +1;
				IF Delta_Shuttle=NUM_SIM_SHUTTLES+2 THEN
					Delta_Shuttle:=0;
				END_IF;
			END_IF;
			IF(gTrakAsm.Command.ShuttleStop) OR VisManual=TRUE THEN
				CntShuttle := 1;
				Step := STOPPING;
			END_IF

			// Error stop
			IF (MC_BR_RoutedMoveVel_AcpTrak_0.Error) THEN
				MC_BR_AsmReset_AcpTrak_0.Execute := TRUE;
				Step := RESET;
			END_IF
			IF NOT(gPartyOn) THEN
				Step:=MANUAL;
			END_IF;
			gVisPower:=TRUE;
	END_CASE

	// Read Assembly status cyclic to Assembly interface
	gTrakAsm.Status.Disabled  := MC_BR_AsmReadStatus_AcpTrak_0.AssemblyDisabled;
	gTrakAsm.Status.Ready     := MC_BR_AsmReadStatus_AcpTrak_0.AssemblyReady;
	gTrakAsm.Status.Homing    := MC_BR_AsmReadStatus_AcpTrak_0.AssemblyHoming;
	gTrakAsm.Status.Stopping  := MC_BR_AsmReadStatus_AcpTrak_0.AssemblyStopping;
	gTrakAsm.Status.ErrorStop := MC_BR_AsmReadStatus_AcpTrak_0.AssemblyErrorStop;

	// Cyclic init functions execute
	MC_BR_AsmPowerOn_AcpTrak_0();
	MC_BR_AsmPowerOn_AcpTrak_0.Execute := FALSE;
	MC_BR_SecAddShuttle_AcpTrak_0();
	MC_BR_SecAddShuttle_AcpTrak_0.Execute := FALSE;
	MC_BR_AsmGetShuttle_AcpTrak_0();
	MC_BR_AsmPowerOff_AcpTrak_0();
	MC_Stop_0();
	MC_BR_RoutedMoveVel_AcpTrak_0();
	MC_BR_AsmReadStatus_AcpTrak_0();
	MC_BR_AsmReset_AcpTrak_0();
	MC_BR_RoutedMoveVel_AcpTrak_0();

	// Timers functions
	TON_Pouring_Top();
	TON_Pouring_Down();
	TON_Delta();
	TON_Capping();

	//Updating values of vel or states with actual data in Visualisation
	gTrakAsm.Command.Power					:=gVisPower;
	gTrakAsm.Command.ShuttleStart			:=VisShuttleStart;
	gTrakAsm.Command.ShuttleStop 			:=VisShuttleStop;
	Pouring_Top_Broken 						:=NOT(VisPouring_Top_Broken);
	Pouring_Down_Broken						:=NOT(VisPouring_Down_Broken);
	Capping_Broken							:=NOT(VisCapping_Broken);
	gTrakAsm.Parameter.Velocity				:=VisVelocity;
	gTrakAsm.Parameter.Acceleration			:=VisAcceleration;
	gTrakAsm.Parameter.Deceleration			:=VisDeceleration;

	CASE gOrder.bottleSize OF
		BOTTLE_SIZE_SMALL:
			TON_Pouring_Down.PT 			:=REAL_TO_TIME(1000*VisPouring_Time_Small);
			TON_Pouring_Top.PT				:=REAL_TO_TIME(1000*VisPouring_Time_Small);
		BOTTLE_SIZE_LARGE:
			TON_Pouring_Down.PT 			:=REAL_TO_TIME(1000*VisPouring_Time_Large);
			TON_Pouring_Top.PT				:=REAL_TO_TIME(1000*VisPouring_Time_Large);
	END_CASE;

	// Handling Broken stations
	IF EDGENEG(Capping_Broken) THEN
		Capping_Comming:=FALSE;
		SvgTranform[2]:=0;
	END_IF;
	IF gVisInput_Broken THEN
		SvgTranform[0]:=0;
	END_IF
	IF NOT (gVisInput_Broken) THEN
		SvgTranform[0]:=2;
	END_IF;
	IF gVisOutput_Broken THEN
		SvgTranform[1]:=0;
	END_IF
	IF NOT (gVisOutput_Broken) THEN
		SvgTranform[1]:=2;
	END_IF;

	IF gVisPower AND gProcessFinished THEN
		ManualEnable:=TRUE;
	ELSE
		ManualEnable:=FALSE;
	END_IF;
					END_PROGRAM

PROGRAM _EXIT
					(* Insert code here *)

	END_PROGRAM
```

### Program Logical/Trak/Vis (IEC)

#### Types.typ
```iecst
TYPE
	Vis_type : 	STRUCT
		Vis : McAcpTrakAssemblyVisData;
		BckgColor : ARRAY[0..2]OF REAL;
	END_STRUCT;
END_TYPE
```

#### Variables.var
```iecst
VAR
	ShuttlesVisibleFalse : BOOL := FALSE;
	pUserData : REFERENCE TO ShuttleUserData_typ;
	SizeofVis : UDINT := 0;
	NumVisShuttle : USINT := 0;
	i : USINT := 0;
	Vizu : Vis_type;
	BlueChangeRate : REAL;
	GreenChangeRate : REAL;
	RedChangeRate : REAL;
	PositionX : ARRAY[0..9] OF REAL;
	PositionY : ARRAY[0..9] OF REAL;
	RotationZ : ARRAY[0..9] OF REAL;
	New_Variable : INT;
END_VAR
```

#### Main.st
```iecst
PROGRAM _INIT

    // size of Vis structure - this value has to be entered in B&R scene viewer (PVI -> Options -> Size)
	SizeofVis := SIZEOF(Vizu);
	// max number of displayed shuttles
	NumVisShuttle := SIZEOF(Vizu.Vis.Shuttle) / SIZEOF(Vizu.Vis.Shuttle[0]);
	FOR i:=0 TO (NumVisShuttle-1) DO
		Vizu.Vis.Shuttle[i].ColorRed     := 1.000;
		Vizu.Vis.Shuttle[i].ColorGreen   := 1.000;
		Vizu.Vis.Shuttle[i].ColorBlue    := 1.000;
	END_FOR;
	Vizu.BckgColor[0] := 0.5;
	Vizu.BckgColor[1] := 0.5;
	Vizu.BckgColor[2] := 0.5;
	RedChangeRate := 0.01;
	GreenChangeRate := 0.05;
	BlueChangeRate := 0.1;
	New_Variable := 1;
END_PROGRAM

PROGRAM _CYCLIC

	IF gPartyOn THEN
		Vizu.BckgColor[0] := Vizu.BckgColor[0] + RedChangeRate;
		IF  Vizu.BckgColor[0] > 1 THEN
			RedChangeRate := -0.01;
		ELSIF Vizu.BckgColor[0] < 0 THEN
			RedChangeRate := 0.01;
		END_IF;

		Vizu.BckgColor[1] := Vizu.BckgColor[1] + GreenChangeRate;

		IF  Vizu.BckgColor[1] > 1 THEN
			GreenChangeRate := -0.05;
		ELSIF Vizu.BckgColor[1] < 0 THEN
			GreenChangeRate := 0.05;
		END_IF;

		Vizu.BckgColor[2] := Vizu.BckgColor[2] + BlueChangeRate;

		IF  Vizu.BckgColor[2] > 1 THEN
			BlueChangeRate := -0.1;
		ELSIF Vizu.BckgColor[2] < 0 THEN
			BlueChangeRate := 0.1;
		END_IF;
	ELSE
		Vizu.BckgColor[0] := 0.5;
		Vizu.BckgColor[1] := 0.5;
		Vizu.BckgColor[2] := 0.5;
	END_IF;

	New_Variable := New_Variable + 1;

	IF New_Variable = 18 THEN
	  New_Variable := 1;
	END_IF;

	FOR i:=0 TO (NumVisShuttle-1) DO
		IF gShuttleMon.Shuttle[i].Available THEN
			Vizu.Vis.Shuttle[i].Available     := 1;
			Vizu.Vis.Shuttle[i].PositionX     := LREAL_TO_REAL(gShuttleMon.Shuttle[i].Position.X);
			Vizu.Vis.Shuttle[i].PositionY     := LREAL_TO_REAL(gShuttleMon.Shuttle[i].Position.Y);
			Vizu.Vis.Shuttle[i].RotationZ     := LREAL_TO_REAL(gShuttleMon.Shuttle[i].Orientation.Angle1);
			Vizu.Vis.Shuttle[i].ExtentToFront := LREAL_TO_REAL(gShuttleMon.Shuttle[i].ExtentToFront);
			Vizu.Vis.Shuttle[i].ExtentToBack  := LREAL_TO_REAL(gShuttleMon.Shuttle[i].ExtentToBack);
			Vizu.Vis.Shuttle[i].Width         := LREAL_TO_REAL(gShuttleMon.Shuttle[i].Width);
			brsitoa(gShuttleMon.Shuttle[i].Index, ADR(Vizu.Vis.Shuttle[i].Text));
			//

			IF gShuttleMon.Shuttle[i].UserData <> 0 THEN
				pUserData ACCESS gShuttleMon.Shuttle[i].UserData;    // access to user data of this shuttle
				IF gShuttleColor[i] = 1 THEN                     // Color is defined with RGB values between 0 and 1
					Vizu.Vis.Shuttle[i].ColorRed     := 0.000;
					Vizu.Vis.Shuttle[i].ColorGreen   := 1.000;
					Vizu.Vis.Shuttle[i].ColorBlue    := 0.000;
				ELSIF gShuttleColor[i] = 2 THEN
					Vizu.Vis.Shuttle[i].ColorRed     := 1.000;
					Vizu.Vis.Shuttle[i].ColorGreen   := 0.000;
					Vizu.Vis.Shuttle[i].ColorBlue    := 0.000;
				ELSIF gShuttleColor[i] = 3 THEN
					Vizu.Vis.Shuttle[i].ColorRed     := 0.000;
					Vizu.Vis.Shuttle[i].ColorGreen   := 0.000;
					Vizu.Vis.Shuttle[i].ColorBlue    := 1.000;
				ELSIF pUserData.Color = 0 THEN
					Vizu.Vis.Shuttle[i].ColorRed     := 1.000;
					Vizu.Vis.Shuttle[i].ColorGreen   := 1.000;
					Vizu.Vis.Shuttle[i].ColorBlue    := 1.000;
				END_IF
			END_IF

		ELSE
			brsmemset(ADR(Vizu.Vis.Shuttle[i]), 0, SIZEOF(Vizu.Vis.Shuttle[0]));  //If the selected shuttle is not available, it will be invisible in the Scene Viewer
		END_IF
	END_FOR
	FOR i:=0 TO 9 DO
		PositionX[i]:=Vizu.Vis.Shuttle[i].PositionX;
		PositionY[i]:=Vizu.Vis.Shuttle[i].PositionX;
		RotationZ[i]:=Vizu.Vis.Shuttle[i].RotationZ;
	END_FOR;

END_PROGRAM
```

### Program Logical/Trak/Recipe

#### Variables.var
```iecst
(*FB's*)
VAR
	MpRecipeXML_0 : MpRecipeXml;
	MpRecipeRegPar_0 : MpRecipeRegPar;
	MpRecipeUI_0 : MpRecipeUI;
END_VAR
(*Structures*)
VAR
	UISetup : MpRecipeUISetupType;
	UIConnect : MpRecipeUIConnectType;
	ClientOrder : Order_type; (*Currently loaded recipe*)
END_VAR
(*IO's*)
VAR
	diErrorReset : BOOL;
END_VAR
(*Other*)
VAR
	WidgetString : ARRAY[0..19] OF STRING[255];
	ErrorMessage : STRING[256];
	Filename : STRING[80];
	i : INT; (*Loop iterator*)
	isError : BOOL;
	PVName : STRING[100];
	Temp : STRING[2]; (*Temporarly stores interator converted to string*)
END_VAR
```

#### Main.st
```iecst
PROGRAM _INIT
	Filename := 'OutFile';
	ErrorMessage := '';
	PVName := 'Recipe:ClientOrder';

	gOrder.bottleSize := 0;
	gOrder.bottlesPerPackage := 0;
	gOrder.drinkColor := 0;
	gOrder.numberOfPackages := 0;

	MpRecipeXML_0.MpLink := ADR(gRecipeXml);
	MpRecipeXML_0.DeviceName := ADR('CF');
	MpRecipeXML_0.FileName := ADR(Filename);
	MpRecipeXML_0.Enable := TRUE;

	MpRecipeRegPar_0.MpLink := ADR(gRecipeXml);
	MpRecipeRegPar_0.PVName := ADR(PVName);
	MpRecipeRegPar_0.Enable := TRUE;

	MpRecipeUI_0.MpLink := ADR(gRecipeXml);
	MpRecipeUI_0.Enable := TRUE;
	UISetup.RecipeListSize:= 20;
	UIConnect.Recipe.Refresh := TRUE;

	MpRecipeUI_0.UISetup := UISetup;
	MpRecipeUI_0.UIConnect := ADR(UIConnect);

END_PROGRAM

PROGRAM _CYCLIC
	MpRecipeXML_0();
	MpRecipeRegPar_0();
	MpRecipeUI_0();

	IF gProcessFinished THEN
		gOrder := ClientOrder;
	END_IF;

	FOR i := 0 TO 19 BY 1 DO
		// delete contents of WidgetString[i]
		WidgetString[i] := DELETE(WidgetString[i], 255, 0);
		IF UIConnect.Recipe.List.Names[i] <> '' THEN

			// convert value of i and store it in Temp
			brsitoa(i, ADR(Temp));

			// Construction of string '{"value":"<i>","text":"<UIConnect.Recipe.List.Names[i]>"}'
			WidgetString[i] := CONCAT(WidgetString[i], '{"value":"');
			WidgetString[i] := CONCAT(WidgetString[i], Temp);
			WidgetString[i] := CONCAT(WidgetString[i], '","text":"');
			WidgetString[i] := CONCAT(WidgetString[i], UIConnect.Recipe.List.Names[i]);
			WidgetString[i] := CONCAT(WidgetString[i], '"}');
		END_IF;
	END_FOR;

	MpRecipeXML_0.ErrorReset := diErrorReset;
	MpRecipeRegPar_0.ErrorReset:= diErrorReset;
	MpRecipeUI_0.ErrorReset := diErrorReset;

	IF MpRecipeXML_0.Error OR MpRecipeRegPar_0.Error OR MpRecipeUI_0.Error THEN
		isError := TRUE;
		IF MpRecipeXML_0.Info.Diag.StatusID.ID = mpRECIPE_ERR_LOAD_WITH_ERRORS
			OR MpRecipeUI_0.Info.Diag.StatusID.ID = mpRECIPE_ERR_LOAD_WITH_ERRORS THEN
			// Damaged XML structure
			ErrorMessage := 'XML structure may be damaged. Check if all tags are correct!';
		ELSIF MpRecipeXML_0.Info.Diag.StatusID.ID = mpRECIPE_ERR_LOAD_DATA
			OR MpRecipeUI_0.Info.Diag.StatusID.ID = mpRECIPE_ERR_LOAD_DATA THEN
			// File is missing
			ErrorMessage := 'The file or XML structure may be missing!';
		ELSIF UIConnect.Recipe.NewFileName = '' AND MpRecipeUI_0.Error THEN
			// Somebody tried to add recipe without new name
			ErrorMessage := 'You must enter new file name!';
		END_IF;
	ELSE
		ErrorMessage := '';
		diErrorReset := FALSE;
		isError := FALSE;
	END_IF;

END_PROGRAM

PROGRAM _EXIT
	MpRecipeXML_0.Enable := FALSE;
	MpRecipeXML_0();

	MpRecipeRegPar_0.Enable := FALSE;
	MpRecipeRegPar_0();

	MpRecipeUI_0.Enable := FALSE;
	MpRecipeUI_0();
END_PROGRAM
```

### Program Logical/Alarms (IEC)

#### Variables.var
```iecst
VAR
	MpAlarmXCore_0 : MpAlarmXCore;
	MpAlarmXHistory_0 : MpAlarmXHistory;
	TrakStop : BOOL;
END_VAR
```

#### Main.st
```iecst
PROGRAM _INIT
	MpAlarmXCore_0.MpLink := ADR(gAlarmXCore);
	MpAlarmXCore_0.Enable := TRUE;

	MpAlarmXHistory_0.MpLink :=ADR(gAlarmXHistory);
	MpAlarmXHistory_0.Enable := TRUE;
END_PROGRAM

PROGRAM _CYCLIC
//	IF EDGEPOS(gdiInstatntStop) THEN
//		MpAlarmXSet(gAlarmXCore, 'InterruptAlarm');
//	END_IF;
//	IF EDGENEG(gdiInstatntStop) THEN
//	  MpAlarmXReset(gAlarmXCore, 'InterruptAlarm');
//	END_IF;

	IF EDGEPOS(TrakStop) THEN
		MpAlarmXSet(gAlarmXCore, 'SuddenlyStopAlarm');
	END_IF;
	IF EDGENEG(TrakStop) THEN
		MpAlarmXReset(gAlarmXCore, 'SuddenlyStopAlarm');
	END_IF;

	MpAlarmXCore_0();
	MpAlarmXHistory_0();
END_PROGRAM

PROGRAM _EXIT
	MpAlarmXCore_0.Enable := FALSE;
	MpAlarmXHistory_0.Enable := FALSE;

	MpAlarmXCore_0();
	MpAlarmXHistory_0();
END_PROGRAM
```

### Program Logical/Recipe (IEC)

#### Types.typ
```iecst
TYPE
	Error_type :
		(
		NO_ERROR,
		ERROR_FILE_MISSING,
		ERROR_WRONG_FILE_NAME,
		ERROR_XML_DAMAGED
		);
END_TYPE
```

#### Variables.var
```iecst
(*FB's*)
VAR
	MpRecipeXML_0 : MpRecipeXml;
	MpRecipeRegPar_0 : MpRecipeRegPar;
	MpRecipeUI_0 : MpRecipeUI;
END_VAR
(*Structures*)
VAR
	UISetup : MpRecipeUISetupType;
	UIConnect : MpRecipeUIConnectType;
	NewRecipe : Order_type;
	ClientOrder : Order_type; (*Currently loaded recipe*)
END_VAR
(*IO's*)
VAR
	diErrorReset : BOOL;
END_VAR
(*Other*)
VAR
	WidgetString : ARRAY[0..19] OF STRING[255];
	Filename : STRING[80];
	i : INT; (*Loop iterator*)
	PVName : STRING[100];
	Temp : STRING[2]; (*Temporarly stores interator converted to string*)
	diLoad : BOOL;
END_VAR
(*Error flags for message box*)
VAR
	ErrorStatus : Error_type := NO_ERROR;
	diAdd : BOOL;
	coffinFlag : BOOL;
END_VAR
```

#### Main.st
```iecst
PROGRAM _INIT
	Filename := 'OutFile';
	PVName := 'Recipe:ClientOrder';

	gOrder.bottleSize := 0;
	gOrder.bottlesPerPackage := 0;
	gOrder.drinkColor := 0;
	gOrder.numberOfPackages := 0;

	NewRecipe.bottlesPerPackage := 0;
	NewRecipe.numberOfPackages := 0;
	NewRecipe.drinkColor := 0;
	NewRecipe.bottleSize := 0;

	MpRecipeXML_0.MpLink := ADR(gRecipeXml);
	MpRecipeXML_0.DeviceName := ADR('CF');
	MpRecipeXML_0.FileName := ADR(Filename);
	MpRecipeXML_0.Enable := TRUE;

	MpRecipeRegPar_0.MpLink := ADR(gRecipeXml);
	MpRecipeRegPar_0.PVName := ADR(PVName);
	MpRecipeRegPar_0.Enable := TRUE;

	MpRecipeUI_0.MpLink := ADR(gRecipeXml);
	MpRecipeUI_0.Enable := TRUE;
	UISetup.RecipeListSize:= 20;
	UIConnect.Recipe.Refresh := TRUE;

	MpRecipeUI_0.UISetup := UISetup;
	MpRecipeUI_0.UIConnect := ADR(UIConnect);

END_PROGRAM

PROGRAM _CYCLIC
	MpRecipeXML_0();
	MpRecipeRegPar_0();
	MpRecipeUI_0();

	IF gProcessFinished AND diLoad THEN
		diLoad := FALSE;
		gOrder := ClientOrder;
		gCurrentRecipeName := UIConnect.Recipe.List.Names[UIConnect.Recipe.List.SelectedIndex];
	END_IF;

	IF UIConnect.New.FileName = 'Death' THEN
		coffinFlag := TRUE;
	ELSE
		coffinFlag := FALSE;
	END_IF;

	IF UIConnect.New.FileName = 'Party' THEN
		gPartyOn := TRUE;
	ELSE
		gPartyOn := FALSE;
	END_IF;

	IF diAdd AND NOT(diLoad) THEN
		ClientOrder := NewRecipe;
		UIConnect.New.Create := TRUE;
		diAdd := FALSE;
		MpRecipeUI_0();
	END_IF;

	IF EDGENEG(UIConnect.New.Create) THEN
		UIConnect.New.FileName := '';
		NewRecipe.bottlesPerPackage := 0;
		NewRecipe.numberOfPackages := 0;
		NewRecipe.drinkColor := 0;
		NewRecipe.bottleSize := 0;

	END_IF;
	UIConnect.Recipe;

	FOR i := 0 TO 19 BY 1 DO
		// delete contents of WidgetString[i]
		WidgetString[i] := DELETE(WidgetString[i], 255, 0);
		IF UIConnect.Recipe.List.Names[i] <> '' THEN

			// convert value of i and store it in Temp
			brsitoa(i, ADR(Temp));

			// Construction of string '{"value":"<i>","text":"<UIConnect.Recipe.List.Names[i]>"}'
			WidgetString[i] := CONCAT(WidgetString[i], '{"value":"');
			WidgetString[i] := CONCAT(WidgetString[i], Temp);
			WidgetString[i] := CONCAT(WidgetString[i], '","text":"');
			WidgetString[i] := CONCAT(WidgetString[i], UIConnect.Recipe.List.Names[i]);
			WidgetString[i] := CONCAT(WidgetString[i], '"}');
		END_IF;
	END_FOR;

	// Error reset handling
	MpRecipeXML_0.ErrorReset := diErrorReset;
	MpRecipeRegPar_0.ErrorReset:= diErrorReset;
	MpRecipeUI_0.ErrorReset := diErrorReset;

	IF MpRecipeXML_0.Error OR MpRecipeRegPar_0.Error OR MpRecipeUI_0.Error THEN
		IF MpRecipeXML_0.Info.Diag.StatusID.ID = mpRECIPE_ERR_LOAD_WITH_ERRORS
			OR MpRecipeUI_0.Info.Diag.StatusID.ID = mpRECIPE_ERR_LOAD_WITH_ERRORS THEN
			// Damaged XML structure
			ErrorStatus := ERROR_XML_DAMAGED;
		ELSIF MpRecipeXML_0.Info.Diag.StatusID.ID = mpRECIPE_ERR_LOAD_DATA
			OR MpRecipeUI_0.Info.Diag.StatusID.ID = mpRECIPE_ERR_LOAD_DATA THEN
			// File is missing
			ErrorStatus := ERROR_FILE_MISSING;
		ELSIF (UIConnect.Recipe.NewFileName = '' OR UIConnect.New.FileName = '') AND MpRecipeUI_0.Error THEN
			// Somebody tried to add recipe without new name
			ErrorStatus := ERROR_WRONG_FILE_NAME;
		END_IF;
	ELSE
		ErrorStatus := NO_ERROR;
		diErrorReset := FALSE;
	END_IF;

END_PROGRAM

PROGRAM _EXIT
	MpRecipeXML_0.Enable := FALSE;
	MpRecipeXML_0();

	MpRecipeRegPar_0.Enable := FALSE;
	MpRecipeRegPar_0();

	MpRecipeUI_0.Enable := FALSE;
	MpRecipeUI_0();
END_PROGRAM
```

### Instruction.txt
```
To run simulaton ACOPOSTrak You need to have Scene Viever 4 and Automation Studio 4.7.3 or higher

Place all of this files (ACOPOSTrak package) at C (path C://ACOPOSTrak)

In Scene Viewer 4:
Online-->PVI-->Options
Task Name : Vis
Variable name : Vizu
Size[bytes] : 10812

Then Connect PVI and OPCUA.

After starting simulation in Automation Studio You can open this link from Your browser (Google Chrome recomended)
http://127.0.0.1:81/index.html?visuId=trakVis
```

### Program Logical/DeltaIn

#### Types.typ
```iecst
TYPE
	StepType :
		(
		Init,
		Power,
		Home,
		Choose,
		WaitShuttle,
		MovePrg,
		Interrupt,
		Stop
		);
END_TYPE
```

#### Variables.var
```iecst
VAR
	GroupPosition : MC_GroupReadActualPosition_15;
	DeltaParameters : MpDelta3AxisParType;
	MpDelta3Axis_0 : MpDelta3Axis;
END_VAR
```

#### Main.st
```iecst
PROGRAM _INIT

	MpDelta3Axis_0.MpLink := ADR(g3AxDeltaA);
	MpDelta3Axis_0.Enable := TRUE;
	MpDelta3Axis_0.Parameters := ADR(DeltaParameters);

	MpDelta3Axis_0.Override := 100.0;
	DeltaParameters.ProgramName := 'RoboticIn.st';    //File stored on FileDevice
	DeltaParameters.Velocity := 5.0;
	DeltaParameters.Acceleration := 50.0;
	Step := Init;
END_PROGRAM

PROGRAM _CYCLIC

	MpDelta3Axis_0();
	IF diStop THEN
		Step:=Stop;
	END_IF;

	CASE Step OF
		Init:
			IF diStart THEN
	  			Step := Power;
			END_IF;
		Power:
			MpDelta3Axis_0.Power := TRUE;
			IF MpDelta3Axis_0.PowerOn THEN
	  			Step:= Home;
			END_IF;
		Home:
			MpDelta3Axis_0.Home := TRUE;
			IF MpDelta3Axis_0.IsHomed THEN
	  			Step := Choose;
			END_IF;
		Choose:
		WaitShuttle:
		MovePrg:
		Interrupt:
		Stop:

	END_CASE;

END_PROGRAM

PROGRAM _EXIT

	MpDelta3Axis_0.Power  := FALSE;
	MpDelta3Axis_0.Home   := FALSE;
	MpDelta3Axis_0.MoveDirect := FALSE;
	MpDelta3Axis_0.MoveLinear := FALSE;
	MpDelta3Axis_0();

	MpDelta3Axis_0.Enable := FALSE;
	MpDelta3Axis_0();

END_PROGRAM
```

### Program Logical/DeltaOut

#### Variables.var
```iecst
VAR
	DeltaParameters : MpDelta3AxisParType;
	MpDelta3Axis_0 : MpDelta3Axis;
END_VAR
```

#### Main.st
```iecst
PROGRAM _INIT

	MpDelta3Axis_0.MpLink := ADR(g3AxDeltaAOut);
	MpDelta3Axis_0.Enable := TRUE;
	MpDelta3Axis_0.Parameters := ADR(DeltaParameters);

	MpDelta3Axis_0.Override := 100.0;

	DeltaParameters.ProgramName := 'Robotic1.st';    //File stored on FileDevice
	DeltaParameters.Velocity := 5.0;
	DeltaParameters.Acceleration := 50.0;

END_PROGRAM

PROGRAM _CYCLIC

	MpDelta3Axis_0();

END_PROGRAM

PROGRAM _EXIT

	MpDelta3Axis_0.Power  := FALSE;
	MpDelta3Axis_0.Home   := FALSE;
	MpDelta3Axis_0.MoveDirect := FALSE;
	MpDelta3Axis_0.MoveLinear := FALSE;
	MpDelta3Axis_0();

	MpDelta3Axis_0.Enable := FALSE;
	MpDelta3Axis_0();

END_PROGRAM
```

### Program Logical/Program

#### Variables.var
```iecst
VAR
	GroupPosition : MC_GroupReadActualPosition_15;
	DeltaParameters : MpDelta3AxisParType;
	MpDelta3Axis_0 : MpDelta3Axis;
END_VAR
```

#### Main.st
```iecst
PROGRAM _INIT

	MpDelta3Axis_0.MpLink := ADR(g3AxDeltaA);
	MpDelta3Axis_0.Enable := TRUE;
	MpDelta3Axis_0.Parameters := ADR(DeltaParameters);

	MpDelta3Axis_0.Override := 100.0;
	DeltaParameters.ProgramName := 'Robotic.st';    //File stored on FileDevice
	DeltaParameters.Velocity := 500.0;
	DeltaParameters.Acceleration := 5000.0;
	DeltaParameters.Deceleration := 5000.0;

	groupReadActualPos.AxesGroup := ADR(g3AxDeltaA);
	groupReadActualPos.Enable := TRUE;
	groupReadActualPos.CoordSystem := 0;

END_PROGRAM

PROGRAM _CYCLIC

	groupReadActualPos();
	MpDelta3Axis_0();

END_PROGRAM

PROGRAM _EXIT

	MpDelta3Axis_0.Power  := FALSE;
	MpDelta3Axis_0.Home   := FALSE;
	MpDelta3Axis_0.MoveDirect := FALSE;
	MpDelta3Axis_0.MoveLinear := FALSE;
	MpDelta3Axis_0();

	MpDelta3Axis_0.Enable := FALSE;
	MpDelta3Axis_0();

END_PROGRAM
```

### Program Logical/Program1

#### Types.typ
```iecst
TYPE
	CoffeeType : 	STRUCT
		Milk : REAL;
		Temperature : REAL;
		Powder : USINT;
		Water : REAL;
		Sugar : USINT;
	END_STRUCT;
END_TYPE
```

#### Variables.var
```iecst
VAR
	s : STRING[80];
	MpRecipeXML_0 : MpRecipeXml;
	Coffee : CoffeeType;
	MpRecipeRegPar_0 : MpRecipeRegPar;
	CF : STRING[80];
	MyFile : STRING[80];
END_VAR
```

#### Main.st
```iecst
PROGRAM _INIT
	(* Insert code here *)
	CF := 'CF';
	MyFile := 'MyFile';
	s := 'Program1:Coffee';
	MpRecipeXML_0.MpLink := ADR(gRecipeXml);
	MpRecipeXML_0.Enable := TRUE;
	MpRecipeXML_0.DeviceName := ADR(CF);
	MpRecipeXML_0.FileName := ADR(MyFile);

	Coffee.Milk := 50;
	Coffee.Powder:= 10;
	Coffee.Sugar :=5;
	Coffee.Temperature := 80;
	Coffee.Water := 250;

	MpRecipeRegPar_0.MpLink := ADR(gRecipeXml);
	MpRecipeRegPar_0.Enable := TRUE;
	MpRecipeRegPar_0.PVName := ADR(s);

END_PROGRAM

PROGRAM _CYCLIC
	(* Insert code here *)
	MpRecipeXML_0();
	MpRecipeRegPar_0();
END_PROGRAM

PROGRAM _EXIT
	(* Insert code here *)

END_PROGRAM
```

### Instruction.txt
```
To run simulaton ACOPOSTrak You need to have Scene Viever 4 and Automation Studio 4.7.3 or higher

Place all of this files (ACOPOSTrak package) at C (path C://ACOPOSTrak)

In Scene Viewer 4:
Online-->PVI-->Options
Task Name : Vis
Variable name : Vizu
Size[bytes] : 10812

Then Connect PVI and OPCUA.

After starting simulation in Automation Studio You can open this link in Your browser (Google Chrome recomended)
http://127.0.0.1:81/index.html?visuId=trakVis
```

### Program Logical/PutTheseFilesIntoCPlease/ACOPOStrak/Robotics

#### RoboticOut3.st
```iecst
VAR CONSTANT
   P1 : McPointType := (Pos:=(X:=0, Y:=200, Z:=-600));
   P2 : McPointType := (Pos:=(X:=0, Y:=200, Z:=-700));
   P3 : McPointType := (Pos:=(X:=150, Y:=-350, Z:=-600));
   P4 : McPointType := (Pos:=(X:=150, Y:=-350, Z:=-700));
END_VAR

PROGRAM _MAIN
 Feedrate(60000);   //move with reduced speed
 PathAcceleration(600000);
 MoveJ(P1);        //move system to point P1
 MoveJ(P2);        //move system to point P2
 WaitTime(1);        //wait for 1 second
 MoveJ(P1);
 MoveJ(P3);        //move back to origin position
 MoveJ(P4);
 WaitTime(1);
 MoveJ(P3);
 MoveJ(P1);        //move system to point P1
END_PROGRAM
```

#### RoboticOut5.st
```iecst
VAR CONSTANT
   P1 : McPointType := (Pos:=(X:=0, Y:=200, Z:=-600));
   P2 : McPointType := (Pos:=(X:=0, Y:=200, Z:=-700));
   P3 : McPointType := (Pos:=(X:=0, Y:=-150, Z:=-600));
   P4 : McPointType := (Pos:=(X:=0, Y:=-150, Z:=-700));
END_VAR

PROGRAM _MAIN
 Feedrate(60000);   //move with reduced speed
 PathAcceleration(600000);
 MoveJ(P1);        //move system to point P1
 MoveJ(P2);        //move system to point P2
 WaitTime(1);        //wait for 1 second
 MoveJ(P1);
 MoveJ(P3);        //move back to origin position
 MoveJ(P4);
 WaitTime(1);
 MoveJ(P3);
 MoveJ(P1);        //move system to point P1
END_PROGRAM
```

#### SI.st
```iecst
VAR CONSTANT
   P1 : McPointType := (Pos:=(X:=200, Y:=200, Z:=-500));
   P2 : McPointType := (Pos:=(X:=200, Y:=200, Z:=-800));
   P3 : McPointType := (Pos:=(X:=200, Y:=-200, Z:=-500));
   P4 : McPointType := (Pos:=(X:=200, Y:=-200, Z:=-800));
   P5 : McPointType := (Pos:=(X:=-200, Y:=200, Z:=-500));
   P6 : McPointType := (Pos:=(X:=-200, Y:=200, Z:=-800));
   P7 : McPointType := (Pos:=(X:=-200, Y:=-200, Z:=-500));
   P8 : McPointType := (Pos:=(X:=-200, Y:=-200, Z:=-800));
END_VAR

PROGRAM _MAIN
 Feedrate(600000);   //move with reduced speed
 PathAcceleration(6000000);
 MoveJ(P1);        //move system to point P1
 MoveJ(P2);        //move system to point P2

 MoveJ(P1);
 MoveJ(P3);        //move back to origin position
 MoveJ(P4);

 MoveJ(P3);
  MoveJ(P5);        //move system to point P1
 MoveJ(P6);        //move system to point P2

 MoveJ(P5);
 MoveJ(P7);        //move back to origin position
 MoveJ(P8);

 MoveJ(P7);
 MoveJ(P1);        //move system to point P1
END_PROGRAM
```

- slnx.sqlite (binary file, 90112 bytes)
### Program Logical/PutTheseFilesIntoCPlease/Robotics
